LIN {X 0,Y 301.762,Z 448.822,A -85,B 0,C 180,E1 -16309.029,E2 -16309.029} C_VEL
LIN {X 0,Y 304.037,Z 439.587,A -85,B 0,C 180,E1 -16311.349,E2 -16311.349} C_VEL
LIN {X 0,Y 306.34,Z 429.711,A -85,B 0,C 180,E1 -16313.412,E2 -16313.412} C_VEL
LIN {X 0,Y 308.97,Z 418.014,A -85,B 0,C 180,E1 -16315.425,E2 -16315.425} C_VEL
LIN {X 0,Y 311.633,Z 405.588,A -85,B 0,C 180,E1 -16317.172,E2 -16317.172} C_VEL
LIN {X 0,Y 314.203,Z 392.482,A -85,B 0,C 180,E1 -16318.669,E2 -16318.669} C_VEL
LIN {X 0,Y 315.459,Z 385.45,A -85,B 0,C 180,E1 -16319.348,E2 -16319.348} C_VEL
LIN {X 0,Y 313.739,Z 373.355,A -85,B 0,C 180,E1 -16320.726,E2 -16320.726} C_VEL
LIN {X 0,Y 310.787,Z 359.836,A -85,B 0,C 180,E1 -16322.156,E2 -16322.156} C_VEL
LIN {X 0,Y 307.358,Z 347.749,A -85,B 0,C 180,E1 -16323.35,E2 -16323.35} C_VEL
LIN {X 0,Y 301.887,Z 332.55,A -85,B 0,C 180,E1 -16324.764,E2 -16324.764} C_VEL
LIN {X 0,Y 298.924,Z 325.57,A -85,B 0,C 180,E1 -16325.394,E2 -16325.394} C_VEL
LIN {X 0,Y 298.745,Z 324.598,A -85,B 0,C 180,E1 -16325.469,E2 -16325.469} C_VEL
LIN {X 0,Y 299.347,Z 320.548,A -85,B 0,C 180,E1 -16329.337,E2 -16329.337} C_VEL
LIN {X 0,Y 299.608,Z 317.074,A -85,B 0,C 180,E1 -16332.863,E2 -16332.863} C_VEL
LIN {X 0,Y 299.433,Z 314.897,A -85,B 0,C 180,E1 -16335.241,E2 -16335.241} C_VEL
LIN {X 0,Y 298.979,Z 311.805,A -85,B 0,C 180,E1 -16338.838,E2 -16338.838} C_VEL
LIN {X 0,Y 298.58,Z 309.054,A -85,B 0,C 180,E1 -16342.267,E2 -16342.267} C_VEL
LIN {X 0,Y 298.413,Z 307.944,A -85,B 0,C 180,E1 -16343.93,E2 -16343.93} C_VEL
LIN {X 0,Y 298.387,Z 307.95,A -85,B 0,C 180,E1 -16347.983,E2 -16347.983} C_VEL
LIN {X 0,Y 298.452,Z 307.939,A -85,B 0,C 180,E1 -16351.903,E2 -16351.903} C_VEL
LIN {X 0,Y 298.479,Z 307.931,A -85,B 0,C 180,E1 -16354.924,E2 -16354.924} C_VEL
LIN {X 0,Y 298.444,Z 307.935,A -85,B 0,C 180,E1 -16359.315,E2 -16359.315} C_VEL
LIN {X 0,Y 298.531,Z 307.922,A -85,B 0,C 180,E1 -16362.179,E2 -16362.179} C_VEL
LIN {X 0,Y 298.586,Z 307.914,A -85,B 0,C 180,E1 -16364.995,E2 -16364.995} C_VEL
LIN {X 0,Y 298.576,Z 307.918,A -85,B 0,C 180,E1 -16369.146,E2 -16369.146} C_VEL
LIN {X 0,Y 298.69,Z 307.902,A -85,B 0,C 180,E1 -16371.884,E2 -16371.884} C_VEL
LIN {X 0,Y 298.634,Z 307.907,A -85,B 0,C 180,E1 -16374.599,E2 -16374.599} C_VEL
LIN {X 0,Y 298.913,Z 307.875,A -85,B 0,C 180,E1 -16378.653,E2 -16378.653} C_VEL
LIN {X 0,Y 298.913,Z 307.878,A -85,B 0,C 180,E1 -16381.347,E2 -16381.347} C_VEL
LIN {X 0,Y 298.635,Z 307.911,A -85,B 0,C 180,E1 -16385.402,E2 -16385.402} C_VEL
LIN {X 0,Y 298.701,Z 307.898,A -85,B 0,C 180,E1 -16388.82,E2 -16388.82} C_VEL
LIN {X 0,Y 298.545,Z 307.924,A -85,B 0,C 180,E1 -16393.616,E2 -16393.616} C_VEL
LIN {X 0,Y 298.542,Z 307.923,A -85,B 0,C 180,E1 -16396.409,E2 -16396.409} C_VEL
LIN {X 0,Y 298.506,Z 307.928,A -85,B 0,C 180,E1 -16399.655,E2 -16399.655} C_VEL
LIN {X 0,Y 298.452,Z 307.934,A -85,B 0,C 180,E1 -16403.598,E2 -16403.598} C_VEL
LIN {X 0,Y 298.481,Z 307.928,A -85,B 0,C 180,E1 -16406.575,E2 -16406.575} C_VEL
LIN {X 0,Y 298.411,Z 307.935,A -85,B 0,C 180,E1 -16409.642,E2 -16409.642} C_VEL
LIN {X 0,Y 298.39,Z 307.937,A -85,B 0,C 180,E1 -16412.801,E2 -16412.801} C_VEL
LIN {X 0,Y 298.442,Z 307.934,A -85,B 0,C 180,E1 -16416.808,E2 -16416.808} C_VEL
LIN {X 0,Y 298.4,Z 307.942,A -85,B 0,C 180,E1 -16419.488,E2 -16419.488} C_VEL
LIN {X 0,Y 298.762,Z 310.457,A -85,B 0,C 180,E1 -16423.179,E2 -16423.179} C_VEL
LIN {X 0,Y 298.971,Z 311.975,A -85,B 0,C 180,E1 -16425.154,E2 -16425.154} C_VEL
LIN {X 0,Y 299.091,Z 315.034,A -85,B 0,C 180,E1 -16428.859,E2 -16428.859} C_VEL
LIN {X 0,Y 298.739,Z 318.083,A -85,B 0,C 180,E1 -16432.291,E2 -16432.291} C_VEL
LIN {X 0,Y 298.531,Z 320.183,A -85,B 0,C 180,E1 -16434.571,E2 -16434.571} C_VEL
LIN {X 0,Y 299.493,Z 323.226,A -85,B 0,C 180,E1 -16434.808,E2 -16434.808} C_VEL
LIN {X 0,Y 304.021,Z 333.557,A -85,B 0,C 180,E1 -16435.807,E2 -16435.807} C_VEL
LIN {X 0,Y 309.067,Z 347.625,A -85,B 0,C 180,E1 -16437.201,E2 -16437.201} C_VEL
LIN {X 0,Y 312.811,Z 361.239,A -85,B 0,C 180,E1 -16438.623,E2 -16438.623} C_VEL
LIN {X 0,Y 315.268,Z 373.146,A -85,B 0,C 180,E1 -16439.956,E2 -16439.956} C_VEL
LIN {X 0,Y 316.015,Z 378.195,A -85,B 0,C 180,E1 -16440.556,E2 -16440.556} C_VEL
LIN {X 0,Y 313.903,Z 390.512,A -85,B 0,C 180,E1 -16441.776,E2 -16441.776} C_VEL
LIN {X 0,Y 311.326,Z 403.463,A -85,B 0,C 180,E1 -16443.343,E2 -16443.343} C_VEL
LIN {X 0,Y 308.75,Z 415.307,A -85,B 0,C 180,E1 -16445.096,E2 -16445.096} C_VEL
LIN {X 0,Y 306.343,Z 426.145,A -85,B 0,C 180,E1 -16447.046,E2 -16447.046} C_VEL
LIN {X 0,Y 303.758,Z 436.69,A -85,B 0,C 180,E1 -16449.34,E2 -16449.34} C_VEL
LIN {X 0,Y 301.665,Z 445.456,A -85,B 0,C 180,E1 -16451.669,E2 -16451.669} C_VEL
LIN {X 0,Y 299.955,Z 452.887,A -85,B 0,C 180,E1 -16454.069,E2 -16454.069} C_VEL
LIN {X 0,Y 298.725,Z 458.754,A -85,B 0,C 180,E1 -16456.393,E2 -16456.393} C_VEL
LIN {X 0,Y 297.61,Z 464.23,A -85,B 0,C 180,E1 -16459.111,E2 -16459.111} C_VEL
LIN {X 0,Y 296.951,Z 468.363,A -85,B 0,C 180,E1 -16461.837,E2 -16461.837} C_VEL
LIN {X 0,Y 296.62,Z 471.267,A -85,B 0,C 180,E1 -16464.562,E2 -16464.562} C_VEL
LIN {X 0,Y 296.531,Z 473.012,A -85,B 0,C 180,E1 -16467.284,E2 -16467.284} C_VEL
LIN {X 0,Y 296.452,Z 473.621,A -85,B 0,C 180,E1 -16470.001,E2 -16470.001} C_VEL
LIN {X 0,Y 296.531,Z 473.052,A -85,B 0,C 180,E1 -16472.717,E2 -16472.717} C_VEL
LIN {X 0,Y 296.667,Z 471.11,A -85,B 0,C 180,E1 -16475.744,E2 -16475.744} C_VEL
LIN {X 0,Y 296.948,Z 468.508,A -85,B 0,C 180,E1 -16478.164,E2 -16478.164} C_VEL
LIN {X 0,Y 297.589,Z 464.424,A -85,B 0,C 180,E1 -16480.891,E2 -16480.891} C_VEL
LIN {X 0,Y 298.694,Z 459.01,A -85,B 0,C 180,E1 -16483.609,E2 -16483.609} C_VEL
LIN {X 0,Y 300.118,Z 452.113,A -85,B 0,C 180,E1 -16486.321,E2 -16486.321} C_VEL
LIN {X 0,Y 302.151,Z 443.505,A -85,B 0,C 180,E1 -16489.004,E2 -16489.004} C_VEL
LIN {X 0,Y 304.328,Z 434.355,A -85,B 0,C 180,E1 -16491.329,E2 -16491.329} C_VEL
LIN {X 0,Y 306.813,Z 424.173,A -85,B 0,C 180,E1 -16493.456,E2 -16493.456} C_VEL
LIN {X 0,Y 309.545,Z 411.912,A -85,B 0,C 180,E1 -16495.555,E2 -16495.555} C_VEL
LIN {X 0,Y 312.17,Z 399.379,A -85,B 0,C 180,E1 -16497.304,E2 -16497.304} C_VEL
LIN {X 0,Y 314.664,Z 387.068,A -85,B 0,C 180,E1 -16498.699,E2 -16498.699} C_VEL
LIN {X 0,Y 316.044,Z 379.083,A -85,B 0,C 180,E1 -16499.464,E2 -16499.464} C_VEL
LIN {X 0,Y 314.514,Z 368.782,A -85,B 0,C 180,E1 -16500.65,E2 -16500.65} C_VEL
LIN {X 0,Y 311.352,Z 355.334,A -85,B 0,C 180,E1 -16502.117,E2 -16502.117} C_VEL
LIN {X 0,Y 307,Z 341.307,A -85,B 0,C 180,E1 -16503.546,E2 -16503.546} C_VEL
LIN {X 0,Y 301.359,Z 327.255,A -85,B 0,C 180,E1 -16504.927,E2 -16504.927} C_VEL
LIN {X 0,Y 298.705,Z 321.182,A -85,B 0,C 180,E1 -16505.492,E2 -16505.492} C_VEL
LIN {X 0,Y 298.545,Z 320.158,A -85,B 0,C 180,E1 -16505.58,E2 -16505.58} C_VEL
LIN {X 0,Y 298.94,Z 316.682,A -85,B 0,C 180,E1 -16509.402,E2 -16509.402} C_VEL
LIN {X 0,Y 299.095,Z 315.081,A -85,B 0,C 180,E1 -16511.243,E2 -16511.243} C_VEL
LIN {X 0,Y 298.986,Z 312.099,A -85,B 0,C 180,E1 -16514.844,E2 -16514.844} C_VEL
LIN {X 0,Y 298.56,Z 309.055,A -85,B 0,C 180,E1 -16518.874,E2 -16518.874} C_VEL
LIN {X 0,Y 298.398,Z 307.943,A -85,B 0,C 180,E1 -16520.512,E2 -16520.512} C_VEL
LIN {X 0,Y 298.418,Z 307.942,A -85,B 0,C 180,E1 -16523.93,E2 -16523.93} C_VEL
LIN {X 0,Y 298.387,Z 307.944,A -85,B 0,C 180,E1 -16527.985,E2 -16527.985} C_VEL
LIN {X 0,Y 298.413,Z 307.939,A -85,B 0,C 180,E1 -16531.899,E2 -16531.899} C_VEL
LIN {X 0,Y 298.439,Z 307.935,A -85,B 0,C 180,E1 -16534.92,E2 -16534.92} C_VEL
LIN {X 0,Y 298.439,Z 307.936,A -85,B 0,C 180,E1 -16539.314,E2 -16539.314} C_VEL
LIN {X 0,Y 298.536,Z 307.924,A -85,B 0,C 180,E1 -16542.179,E2 -16542.179} C_VEL
LIN {X 0,Y 298.547,Z 307.918,A -85,B 0,C 180,E1 -16543.586,E2 -16543.586} C_VEL
LIN {X 0,Y 297.935,Z 307.998,A -85,B 0,C 180,E1 -16544.713,E2 -16544.713} C_VEL
LIN {X 0,Y 295.079,Z 308.355,A -85,B 0,C 180,E1 -16546.547,E2 -16546.547} C_VEL
LIN {X 0,Y 292.632,Z 308.658,A -85,B 0,C 180,E1 -16548.036,E2 -16548.036} C_VEL
LIN {X 0,Y 291.598,Z 308.789,A -85,B 0,C 180,E1 -16549.19,E2 -16549.19} C_VEL
LIN {X 0,Y 291.525,Z 308.794,A -85,B 0,C 180,E1 -16549.581,E2 -16549.581} C_VEL
LIN {X 0,Y 291.65,Z 308.78,A -85,B 0,C 180,E1 -16551.687,E2 -16551.687} C_VEL
LIN {X 0,Y 291.607,Z 308.787,A -85,B 0,C 180,E1 -16554.468,E2 -16554.468} C_VEL
LIN {X 0,Y 291.885,Z 308.753,A -85,B 0,C 180,E1 -16558.62,E2 -16558.62} C_VEL
LIN {X 0,Y 291.884,Z 308.752,A -85,B 0,C 180,E1 -16561.38,E2 -16561.38} C_VEL
LIN {X 0,Y 291.607,Z 308.786,A -85,B 0,C 180,E1 -16565.532,E2 -16565.532} C_VEL
LIN {X 0,Y 291.665,Z 308.779,A -85,B 0,C 180,E1 -16568.91,E2 -16568.91} C_VEL
LIN {X 0,Y 291.516,Z 308.799,A -85,B 0,C 180,E1 -16572.531,E2 -16572.531} C_VEL
LIN {X 0,Y 291.554,Z 308.795,A -85,B 0,C 180,E1 -16575.376,E2 -16575.376} C_VEL
LIN {X 0,Y 291.45,Z 308.808,A -85,B 0,C 180,E1 -16579.875,E2 -16579.875} C_VEL
LIN {X 0,Y 291.381,Z 308.815,A -85,B 0,C 180,E1 -16584.207,E2 -16584.207} C_VEL
LIN {X 0,Y 291.418,Z 308.813,A -85,B 0,C 180,E1 -16587.272,E2 -16587.272} C_VEL
LIN {X 0,Y 291.333,Z 308.827,A -85,B 0,C 180,E1 -16590.437,E2 -16590.437} C_VEL
LIN {X 0,Y 291.343,Z 308.829,A -85,B 0,C 180,E1 -16593.698,E2 -16593.698} C_VEL
LIN {X 0,Y 291.36,Z 308.828,A -85,B 0,C 180,E1 -16595.374,E2 -16595.374} C_VEL
LIN {X 0,Y 291.722,Z 311.173,A -85,B 0,C 180,E1 -16598.783,E2 -16598.783} C_VEL
LIN {X 0,Y 292.146,Z 314.013,A -85,B 0,C 180,E1 -16602.344,E2 -16602.344} C_VEL
LIN {X 0,Y 292.518,Z 317.273,A -85,B 0,C 180,E1 -16606.118,E2 -16606.118} C_VEL
LIN {X 0,Y 292.391,Z 320.487,A -85,B 0,C 180,E1 -16609.535,E2 -16609.535} C_VEL
LIN {X 0,Y 291.975,Z 323.962,A -85,B 0,C 180,E1 -16613.004,E2 -16613.004} C_VEL
LIN {X 0,Y 291.891,Z 324.512,A -85,B 0,C 180,E1 -16613.537,E2 -16613.537} C_VEL
LIN {X 0,Y 292.88,Z 327.696,A -85,B 0,C 180,E1 -16613.802,E2 -16613.802} C_VEL
LIN {X 0,Y 298.34,Z 340.78,A -85,B 0,C 180,E1 -16615.093,E2 -16615.093} C_VEL
LIN {X 0,Y 302.962,Z 355.274,A -85,B 0,C 180,E1 -16616.553,E2 -16616.553} C_VEL
LIN {X 0,Y 306.134,Z 368.142,A -85,B 0,C 180,E1 -16617.937,E2 -16617.937} C_VEL
LIN {X 0,Y 308.432,Z 381.307,A -85,B 0,C 180,E1 -16619.454,E2 -16619.454} C_VEL
LIN {X 0,Y 309.086,Z 386.746,A -85,B 0,C 180,E1 -16620.115,E2 -16620.115} C_VEL
LIN {X 0,Y 306.669,Z 399.186,A -85,B 0,C 180,E1 -16621.419,E2 -16621.419} C_VEL
LIN {X 0,Y 303.725,Z 412.723,A -85,B 0,C 180,E1 -16623.178,E2 -16623.178} C_VEL
LIN {X 0,Y 300.907,Z 424.901,A -85,B 0,C 180,E1 -16625.139,E2 -16625.139} C_VEL
LIN {X 0,Y 298.453,Z 435.156,A -85,B 0,C 180,E1 -16627.143,E2 -16627.143} C_VEL
LIN {X 0,Y 295.925,Z 445.11,A -85,B 0,C 180,E1 -16629.494,E2 -16629.494} C_VEL
LIN {X 0,Y 293.899,Z 453.404,A -85,B 0,C 180,E1 -16631.888,E2 -16631.888} C_VEL
LIN {X 0,Y 292.116,Z 461.195,A -85,B 0,C 180,E1 -16634.654,E2 -16634.654} C_VEL
LIN {X 0,Y 290.835,Z 467.392,A -85,B 0,C 180,E1 -16637.438,E2 -16637.438} C_VEL
LIN {X 0,Y 290.016,Z 472.185,A -85,B 0,C 180,E1 -16640.233,E2 -16640.233} C_VEL
LIN {X 0,Y 289.567,Z 475.696,A -85,B 0,C 180,E1 -16643.029,E2 -16643.029} C_VEL
LIN {X 0,Y 289.374,Z 478.005,A -85,B 0,C 180,E1 -16645.821,E2 -16645.821} C_VEL
LIN {X 0,Y 289.368,Z 479.166,A -85,B 0,C 180,E1 -16648.608,E2 -16648.608} C_VEL
LIN {X 0,Y 289.368,Z 479.163,A -85,B 0,C 180,E1 -16651.391,E2 -16651.391} C_VEL
LIN {X 0,Y 289.376,Z 477.989,A -85,B 0,C 180,E1 -16654.178,E2 -16654.178} C_VEL
LIN {X 0,Y 289.566,Z 475.67,A -85,B 0,C 180,E1 -16656.97,E2 -16656.97} C_VEL
LIN {X 0,Y 290.015,Z 472.154,A -85,B 0,C 180,E1 -16659.766,E2 -16659.766} C_VEL
LIN {X 0,Y 290.833,Z 467.353,A -85,B 0,C 180,E1 -16662.561,E2 -16662.561} C_VEL
LIN {X 0,Y 292.124,Z 461.135,A -85,B 0,C 180,E1 -16665.345,E2 -16665.345} C_VEL
LIN {X 0,Y 293.895,Z 453.328,A -85,B 0,C 180,E1 -16668.111,E2 -16668.111} C_VEL
LIN {X 0,Y 295.913,Z 445.024,A -85,B 0,C 180,E1 -16670.506,E2 -16670.506} C_VEL
LIN {X 0,Y 298.5,Z 435.019,A -85,B 0,C 180,E1 -16672.859,E2 -16672.859} C_VEL
LIN {X 0,Y 300.901,Z 424.786,A -85,B 0,C 180,E1 -16674.86,E2 -16674.86} C_VEL
LIN {X 0,Y 303.701,Z 412.587,A -85,B 0,C 180,E1 -16676.823,E2 -16676.823} C_VEL
LIN {X 0,Y 306.657,Z 399.002,A -85,B 0,C 180,E1 -16678.581,E2 -16678.581} C_VEL
LIN {X 0,Y 309.046,Z 386.658,A -85,B 0,C 180,E1 -16679.873,E2 -16679.873} C_VEL
LIN {X 0,Y 307.37,Z 374.793,A -85,B 0,C 180,E1 -16681.289,E2 -16681.289} C_VEL
LIN {X 0,Y 304.337,Z 360.53,A -85,B 0,C 180,E1 -16682.864,E2 -16682.864} C_VEL
LIN {X 0,Y 300.046,Z 345.896,A -85,B 0,C 180,E1 -16684.371,E2 -16684.371} C_VEL
LIN {X 0,Y 295.025,Z 332.512,A -85,B 0,C 180,E1 -16685.692,E2 -16685.692} C_VEL
LIN {X 0,Y 292.068,Z 325.637,A -85,B 0,C 180,E1 -16686.35,E2 -16686.35} C_VEL
LIN {X 0,Y 291.867,Z 324.527,A -85,B 0,C 180,E1 -16686.427,E2 -16686.427} C_VEL
LIN {X 0,Y 292.326,Z 321.204,A -85,B 0,C 180,E1 -16689.706,E2 -16689.706} C_VEL
LIN {X 0,Y 292.53,Z 318.735,A -85,B 0,C 180,E1 -16692.274,E2 -16692.274} C_VEL
LIN {X 0,Y 292.362,Z 315.557,A -85,B 0,C 180,E1 -16695.804,E2 -16695.804} C_VEL
LIN {X 0,Y 291.889,Z 312.541,A -85,B 0,C 180,E1 -16699.451,E2 -16699.451} C_VEL
LIN {X 0,Y 291.521,Z 309.849,A -85,B 0,C 180,E1 -16702.937,E2 -16702.937} C_VEL
LIN {X 0,Y 291.356,Z 308.824,A -85,B 0,C 180,E1 -16704.625,E2 -16704.625} C_VEL
LIN {X 0,Y 291.364,Z 308.825,A -85,B 0,C 180,E1 -16707.95,E2 -16707.95} C_VEL
LIN {X 0,Y 291.371,Z 308.82,A -85,B 0,C 180,E1 -16711.157,E2 -16711.157} C_VEL
LIN {X 0,Y 291.41,Z 308.812,A -85,B 0,C 180,E1 -16714.271,E2 -16714.271} C_VEL
LIN {X 0,Y 291.375,Z 308.817,A -85,B 0,C 180,E1 -16717.299,E2 -16717.299} C_VEL
LIN {X 0,Y 291.452,Z 308.804,A -85,B 0,C 180,E1 -16720.27,E2 -16720.27} C_VEL
LIN {X 0,Y 291.534,Z 308.794,A -85,B 0,C 180,E1 -16724.634,E2 -16724.634} C_VEL
LIN {X 0,Y 291.522,Z 308.796,A -85,B 0,C 180,E1 -16728.88,E2 -16728.88} C_VEL
LIN {X 0,Y 291.644,Z 308.78,A -85,B 0,C 180,E1 -16731.687,E2 -16731.687} C_VEL
LIN {X 0,Y 291.602,Z 308.783,A -85,B 0,C 180,E1 -16734.468,E2 -16734.468} C_VEL
LIN {X 0,Y 291.88,Z 308.751,A -85,B 0,C 180,E1 -16738.62,E2 -16738.62} C_VEL
LIN {X 0,Y 291.88,Z 308.754,A -85,B 0,C 180,E1 -16741.38,E2 -16741.38} C_VEL
LIN {X 0,Y 291.642,Z 308.78,A -85,B 0,C 180,E1 -16746.533,E2 -16746.533} C_VEL
LIN {X 0,Y 291.561,Z 308.793,A -85,B 0,C 180,E1 -16749.714,E2 -16749.714} C_VEL
LIN {X 0,Y 291.515,Z 308.796,A -85,B 0,C 180,E1 -16753.951,E2 -16753.951} C_VEL
LIN {X 0,Y 291.481,Z 308.802,A -85,B 0,C 180,E1 -16756.818,E2 -16756.818} C_VEL
LIN {X 0,Y 291.445,Z 308.806,A -85,B 0,C 180,E1 -16759.875,E2 -16759.875} C_VEL
LIN {X 0,Y 291.395,Z 308.814,A -85,B 0,C 180,E1 -16764.206,E2 -16764.206} C_VEL
LIN {X 0,Y 291.414,Z 308.808,A -85,B 0,C 180,E1 -16767.273,E2 -16767.273} C_VEL
LIN {X 0,Y 291.329,Z 308.817,A -85,B 0,C 180,E1 -16770.438,E2 -16770.438} C_VEL
LIN {X 0,Y 291.339,Z 308.816,A -85,B 0,C 180,E1 -16773.699,E2 -16773.699} C_VEL
LIN {X 0,Y 291.371,Z 308.815,A -85,B 0,C 180,E1 -16777.255,E2 -16777.255} C_VEL
LIN {X 0,Y 291.398,Z 309.016,A -85,B 0,C 180,E1 -16779.488,E2 -16779.488} C_VEL
LIN {X 0,Y 291.808,Z 312.06,A -85,B 0,C 180,E1 -16783.738,E2 -16783.738} C_VEL
LIN {X 0,Y 292.004,Z 313.967,A -85,B 0,C 180,E1 -16786.224,E2 -16786.224} C_VEL
LIN {X 0,Y 292.003,Z 316.637,A -85,B 0,C 180,E1 -16789.472,E2 -16789.472} C_VEL
LIN {X 0,Y 291.615,Z 320.296,A -85,B 0,C 180,E1 -16793.606,E2 -16793.606} C_VEL
LIN {X 0,Y 292.49,Z 323.161,A -85,B 0,C 180,E1 -16793.829,E2 -16793.829} C_VEL
LIN {X 0,Y 293.765,Z 325.811,A -85,B 0,C 180,E1 -16794.104,E2 -16794.104} C_VEL
LIN {X 0,Y 299.181,Z 338.663,A -85,B 0,C 180,E1 -16795.426,E2 -16795.426} C_VEL
LIN {X 0,Y 303.595,Z 351.639,A -85,B 0,C 180,E1 -16796.792,E2 -16796.792} C_VEL
LIN {X 0,Y 307.308,Z 366.226,A -85,B 0,C 180,E1 -16798.417,E2 -16798.417} C_VEL
LIN {X 0,Y 309.462,Z 378.455,A -85,B 0,C 180,E1 -16799.888,E2 -16799.888} C_VEL
LIN {X 0,Y 309.443,Z 381.11,A -85,B 0,C 180,E1 -16800.175,E2 -16800.175} C_VEL
LIN {X 0,Y 306.792,Z 394.787,A -85,B 0,C 180,E1 -16801.62,E2 -16801.62} C_VEL
LIN {X 0,Y 304.255,Z 407.042,A -85,B 0,C 180,E1 -16803.23,E2 -16803.23} C_VEL
LIN {X 0,Y 301.43,Z 419.251,A -85,B 0,C 180,E1 -16805.187,E2 -16805.187} C_VEL
LIN {X 0,Y 298.988,Z 429.465,A -85,B 0,C 180,E1 -16807.18,E2 -16807.18} C_VEL
LIN {X 0,Y 296.42,Z 439.461,A -85,B 0,C 180,E1 -16809.531,E2 -16809.531} C_VEL
LIN {X 0,Y 294.303,Z 447.752,A -85,B 0,C 180,E1 -16811.915,E2 -16811.915} C_VEL
LIN {X 0,Y 292.733,Z 454.42,A -85,B 0,C 180,E1 -16814.245,E2 -16814.245} C_VEL
LIN {X 0,Y 291.435,Z 460.32,A -85,B 0,C 180,E1 -16816.757,E2 -16816.757} C_VEL
LIN {X 0,Y 290.398,Z 465.467,A -85,B 0,C 180,E1 -16819.543,E2 -16819.543} C_VEL
LIN {X 0,Y 289.895,Z 468.433,A -85,B 0,C 180,E1 -16821.637,E2 -16821.637} C_VEL
LIN {X 0,Y 289.556,Z 471.336,A -85,B 0,C 180,E1 -16824.429,E2 -16824.429} C_VEL
LIN {X 0,Y 289.437,Z 473.081,A -85,B 0,C 180,E1 -16827.217,E2 -16827.217} C_VEL
LIN {X 0,Y 289.372,Z 473.69,A -85,B 0,C 180,E1 -16830.001,E2 -16830.001} C_VEL
LIN {X 0,Y 289.437,Z 473.121,A -85,B 0,C 180,E1 -16832.784,E2 -16832.784} C_VEL
LIN {X 0,Y 289.587,Z 471.317,A -85,B 0,C 180,E1 -16835.713,E2 -16835.713} C_VEL
LIN {X 0,Y 289.892,Z 468.577,A -85,B 0,C 180,E1 -16838.364,E2 -16838.364} C_VEL
LIN {X 0,Y 290.571,Z 464.492,A -85,B 0,C 180,E1 -16841.157,E2 -16841.157} C_VEL
LIN {X 0,Y 291.752,Z 459.078,A -85,B 0,C 180,E1 -16843.939,E2 -16843.939} C_VEL
LIN {X 0,Y 293.25,Z 452.181,A -85,B 0,C 180,E1 -16846.714,E2 -16846.714} C_VEL
LIN {X 0,Y 295.385,Z 443.573,A -85,B 0,C 180,E1 -16849.457,E2 -16849.457} C_VEL
LIN {X 0,Y 297.701,Z 434.422,A -85,B 0,C 180,E1 -16851.828,E2 -16851.828} C_VEL
LIN {X 0,Y 300.112,Z 424.883,A -85,B 0,C 180,E1 -16853.875,E2 -16853.875} C_VEL
LIN {X 0,Y 302.884,Z 413.041,A -85,B 0,C 180,E1 -16855.974,E2 -16855.974} C_VEL
LIN {X 0,Y 305.616,Z 400.724,A -85,B 0,C 180,E1 -16857.754,E2 -16857.754} C_VEL
LIN {X 0,Y 308.372,Z 387.5,A -85,B 0,C 180,E1 -16859.296,E2 -16859.296} C_VEL
LIN {X 0,Y 309.582,Z 380.809,A -85,B 0,C 180,E1 -16859.963,E2 -16859.963} C_VEL
LIN {X 0,Y 309.141,Z 376.231,A -85,B 0,C 180,E1 -16860.503,E2 -16860.503} C_VEL
LIN {X 0,Y 306.677,Z 363.447,A -85,B 0,C 180,E1 -16862.014,E2 -16862.014} C_VEL
LIN {X 0,Y 303.174,Z 350.218,A -85,B 0,C 180,E1 -16863.474,E2 -16863.474} C_VEL
LIN {X 0,Y 298.502,Z 336.794,A -85,B 0,C 180,E1 -16864.892,E2 -16864.892} C_VEL
LIN {X 0,Y 292.91,Z 323.875,A -85,B 0,C 180,E1 -16866.212,E2 -16866.212} C_VEL
LIN {X 0,Y 291.78,Z 321.283,A -85,B 0,C 180,E1 -16866.466,E2 -16866.466} C_VEL
LIN {X 0,Y 291.587,Z 320.238,A -85,B 0,C 180,E1 -16866.567,E2 -16866.567} C_VEL
LIN {X 0,Y 292.007,Z 316.769,A -85,B 0,C 180,E1 -16870.529,E2 -16870.529} C_VEL
LIN {X 0,Y 292.011,Z 313.698,A -85,B 0,C 180,E1 -16874.263,E2 -16874.263} C_VEL
LIN {X 0,Y 291.684,Z 311.211,A -85,B 0,C 180,E1 -16877.573,E2 -16877.573} C_VEL
LIN {X 0,Y 291.351,Z 308.821,A -85,B 0,C 180,E1 -16881.158,E2 -16881.158} C_VEL
LIN {X 0,Y 291.361,Z 308.82,A -85,B 0,C 180,E1 -16884.626,E2 -16884.626} C_VEL
LIN {X 0,Y 291.365,Z 308.818,A -85,B 0,C 180,E1 -16887.95,E2 -16887.95} C_VEL
LIN {X 0,Y 291.343,Z 308.819,A -85,B 0,C 180,E1 -16891.154,E2 -16891.154} C_VEL
LIN {X 0,Y 291.359,Z 308.819,A -85,B 0,C 180,E1 -16894.266,E2 -16894.266} C_VEL
LIN {X 0,Y 291.371,Z 308.814,A -85,B 0,C 180,E1 -16897.298,E2 -16897.298} C_VEL
LIN {X 0,Y 291.457,Z 308.802,A -85,B 0,C 180,E1 -16900.27,E2 -16900.27} C_VEL
LIN {X 0,Y 291.555,Z 308.791,A -85,B 0,C 180,E1 -16904.624,E2 -16904.624} C_VEL
LIN {X 0,Y 291.527,Z 308.797,A -85,B 0,C 180,E1 -16908.88,E2 -16908.88} C_VEL
LIN {X 0,Y 291.525,Z 308.794,A -85,B 0,C 180,E1 -16909.581,E2 -16909.581} C_VEL
LIN {X 0,Y 290.885,Z 308.878,A -85,B 0,C 180,E1 -16910.735,E2 -16910.735} C_VEL
LIN {X 0,Y 288.039,Z 309.232,A -85,B 0,C 180,E1 -16912.615,E2 -16912.615} C_VEL
LIN {X 0,Y 285.613,Z 309.535,A -85,B 0,C 180,E1 -16914.141,E2 -16914.141} C_VEL
LIN {X 0,Y 284.579,Z 309.662,A -85,B 0,C 180,E1 -16915.323,E2 -16915.323} C_VEL
LIN {X 0,Y 284.499,Z 309.672,A -85,B 0,C 180,E1 -16915.724,E2 -16915.724} C_VEL
LIN {X 0,Y 284.852,Z 309.629,A -85,B 0,C 180,E1 -16918.586,E2 -16918.586} C_VEL
LIN {X 0,Y 284.851,Z 309.628,A -85,B 0,C 180,E1 -16921.414,E2 -16921.414} C_VEL
LIN {X 0,Y 284.575,Z 309.662,A -85,B 0,C 180,E1 -16925.669,E2 -16925.669} C_VEL
LIN {X 0,Y 284.606,Z 309.659,A -85,B 0,C 180,E1 -16928.98,E2 -16928.98} C_VEL
LIN {X 0,Y 284.473,Z 309.676,A -85,B 0,C 180,E1 -16932.847,E2 -16932.847} C_VEL
LIN {X 0,Y 284.486,Z 309.674,A -85,B 0,C 180,E1 -16935.768,E2 -16935.768} C_VEL
LIN {X 0,Y 284.376,Z 309.688,A -85,B 0,C 180,E1 -16940.242,E2 -16940.242} C_VEL
LIN {X 0,Y 284.336,Z 309.692,A -85,B 0,C 180,E1 -16944.847,E2 -16944.847} C_VEL
LIN {X 0,Y 284.327,Z 309.696,A -85,B 0,C 180,E1 -16948.011,E2 -16948.011} C_VEL
LIN {X 0,Y 284.292,Z 309.705,A -85,B 0,C 180,E1 -16951.275,E2 -16951.275} C_VEL
LIN {X 0,Y 284.308,Z 309.706,A -85,B 0,C 180,E1 -16954.649,E2 -16954.649} C_VEL
LIN {X 0,Y 284.66,Z 311.954,A -85,B 0,C 180,E1 -16958.114,E2 -16958.114} C_VEL
LIN {X 0,Y 285.148,Z 315.206,A -85,B 0,C 180,E1 -16962.32,E2 -16962.32} C_VEL
LIN {X 0,Y 285.476,Z 317.895,A -85,B 0,C 180,E1 -16965.556,E2 -16965.556} C_VEL
LIN {X 0,Y 285.461,Z 320.418,A -85,B 0,C 180,E1 -16968.338,E2 -16968.338} C_VEL
LIN {X 0,Y 285.079,Z 324.014,A -85,B 0,C 180,E1 -16972.082,E2 -16972.082} C_VEL
LIN {X 0,Y 285.04,Z 324.631,A -85,B 0,C 180,E1 -16972.536,E2 -16972.536} C_VEL
LIN {X 0,Y 286.07,Z 327.739,A -85,B 0,C 180,E1 -16972.801,E2 -16972.801} C_VEL
LIN {X 0,Y 287.425,Z 330.751,A -85,B 0,C 180,E1 -16973.115,E2 -16973.115} C_VEL
LIN {X 0,Y 293.007,Z 344.703,A -85,B 0,C 180,E1 -16974.586,E2 -16974.586} C_VEL
LIN {X 0,Y 297.212,Z 358.54,A -85,B 0,C 180,E1 -16976.064,E2 -16976.064} C_VEL
LIN {X 0,Y 300.11,Z 370.919,A -85,B 0,C 180,E1 -16977.463,E2 -16977.463} C_VEL
LIN {X 0,Y 302.178,Z 383.779,A -85,B 0,C 180,E1 -16979.031,E2 -16979.031} C_VEL
LIN {X 0,Y 302.642,Z 387.691,A -85,B 0,C 180,E1 -16979.534,E2 -16979.534} C_VEL
LIN {X 0,Y 300.137,Z 400.444,A -85,B 0,C 180,E1 -16980.93,E2 -16980.93} C_VEL
LIN {X 0,Y 297.397,Z 412.657,A -85,B 0,C 180,E1 -16982.56,E2 -16982.56} C_VEL
LIN {X 0,Y 294.428,Z 424.834,A -85,B 0,C 180,E1 -16984.554,E2 -16984.554} C_VEL
LIN {X 0,Y 291.787,Z 435.391,A -85,B 0,C 180,E1 -16986.663,E2 -16986.663} C_VEL
LIN {X 0,Y 289.205,Z 445.042,A -85,B 0,C 180,E1 -16988.995,E2 -16988.995} C_VEL
LIN {X 0,Y 287.112,Z 453.336,A -85,B 0,C 180,E1 -16991.445,E2 -16991.445} C_VEL
LIN {X 0,Y 285.19,Z 461.126,A -85,B 0,C 180,E1 -16994.271,E2 -16994.271} C_VEL
LIN {X 0,Y 283.874,Z 467.324,A -85,B 0,C 180,E1 -16997.125,E2 -16997.125} C_VEL
LIN {X 0,Y 282.971,Z 472.116,A -85,B 0,C 180,E1 -16999.988,E2 -16999.988} C_VEL
LIN {X 0,Y 282.487,Z 475.627,A -85,B 0,C 180,E1 -17002.854,E2 -17002.854} C_VEL
LIN {X 0,Y 282.284,Z 477.936,A -85,B 0,C 180,E1 -17005.716,E2 -17005.716} C_VEL
LIN {X 0,Y 282.293,Z 479.097,A -85,B 0,C 180,E1 -17008.573,E2 -17008.573} C_VEL
LIN {X 0,Y 282.293,Z 479.094,A -85,B 0,C 180,E1 -17011.426,E2 -17011.426} C_VEL
LIN {X 0,Y 282.286,Z 477.92,A -85,B 0,C 180,E1 -17014.283,E2 -17014.283} C_VEL
LIN {X 0,Y 282.487,Z 475.6,A -85,B 0,C 180,E1 -17017.145,E2 -17017.145} C_VEL
LIN {X 0,Y 282.97,Z 472.084,A -85,B 0,C 180,E1 -17020.011,E2 -17020.011} C_VEL
LIN {X 0,Y 283.872,Z 467.282,A -85,B 0,C 180,E1 -17022.874,E2 -17022.874} C_VEL
LIN {X 0,Y 285.197,Z 461.064,A -85,B 0,C 180,E1 -17025.727,E2 -17025.727} C_VEL
LIN {X 0,Y 287.106,Z 453.256,A -85,B 0,C 180,E1 -17028.555,E2 -17028.555} C_VEL
LIN {X 0,Y 289.198,Z 444.952,A -85,B 0,C 180,E1 -17031.004,E2 -17031.004} C_VEL
LIN {X 0,Y 291.866,Z 435.101,A -85,B 0,C 180,E1 -17033.373,E2 -17033.373} C_VEL
LIN {X 0,Y 294.419,Z 424.714,A -85,B 0,C 180,E1 -17035.446,E2 -17035.446} C_VEL
LIN {X 0,Y 297.357,Z 412.515,A -85,B 0,C 180,E1 -17037.443,E2 -17037.443} C_VEL
LIN {X 0,Y 300.423,Z 398.928,A -85,B 0,C 180,E1 -17039.231,E2 -17039.231} C_VEL
LIN {X 0,Y 302.571,Z 387.799,A -85,B 0,C 180,E1 -17040.431,E2 -17040.431} C_VEL
LIN {X 0,Y 300.818,Z 375.352,A -85,B 0,C 180,E1 -17041.987,E2 -17041.987} C_VEL
LIN {X 0,Y 298.205,Z 362.464,A -85,B 0,C 180,E1 -17043.472,E2 -17043.472} C_VEL
LIN {X 0,Y 294.034,Z 348.026,A -85,B 0,C 180,E1 -17045.05,E2 -17045.05} C_VEL
LIN {X 0,Y 289.483,Z 335.708,A -85,B 0,C 180,E1 -17046.339,E2 -17046.339} C_VEL
LIN {X 0,Y 285.967,Z 327.591,A -85,B 0,C 180,E1 -17047.181,E2 -17047.181} C_VEL
LIN {X 0,Y 284.978,Z 324.45,A -85,B 0,C 180,E1 -17047.452,E2 -17047.452} C_VEL
LIN {X 0,Y 285.341,Z 321.744,A -85,B 0,C 180,E1 -17050.223,E2 -17050.223} C_VEL
LIN {X 0,Y 285.486,Z 318.652,A -85,B 0,C 180,E1 -17053.573,E2 -17053.573} C_VEL
LIN {X 0,Y 285.296,Z 316.232,A -85,B 0,C 180,E1 -17056.39,E2 -17056.39} C_VEL
LIN {X 0,Y 284.825,Z 313.279,A -85,B 0,C 180,E1 -17060.093,E2 -17060.093} C_VEL
LIN {X 0,Y 284.433,Z 310.657,A -85,B 0,C 180,E1 -17063.629,E2 -17063.629} C_VEL
LIN {X 0,Y 284.303,Z 309.703,A -85,B 0,C 180,E1 -17065.35,E2 -17065.35} C_VEL
LIN {X 0,Y 284.288,Z 309.706,A -85,B 0,C 180,E1 -17068.725,E2 -17068.725} C_VEL
LIN {X 0,Y 284.39,Z 309.688,A -85,B 0,C 180,E1 -17072.826,E2 -17072.826} C_VEL
LIN {X 0,Y 284.36,Z 309.689,A -85,B 0,C 180,E1 -17076.707,E2 -17076.707} C_VEL
LIN {X 0,Y 284.397,Z 309.685,A -85,B 0,C 180,E1 -17081.261,E2 -17081.261} C_VEL
LIN {X 0,Y 284.472,Z 309.675,A -85,B 0,C 180,E1 -17084.469,E2 -17084.469} C_VEL
LIN {X 0,Y 284.476,Z 309.673,A -85,B 0,C 180,E1 -17088.601,E2 -17088.601} C_VEL
LIN {X 0,Y 284.601,Z 309.656,A -85,B 0,C 180,E1 -17091.48,E2 -17091.48} C_VEL
LIN {X 0,Y 284.571,Z 309.658,A -85,B 0,C 180,E1 -17094.331,E2 -17094.331} C_VEL
LIN {X 0,Y 284.846,Z 309.626,A -85,B 0,C 180,E1 -17098.586,E2 -17098.586} C_VEL
LIN {X 0,Y 284.846,Z 309.631,A -85,B 0,C 180,E1 -17101.414,E2 -17101.414} C_VEL
LIN {X 0,Y 284.591,Z 309.658,A -85,B 0,C 180,E1 -17106.55,E2 -17106.55} C_VEL
LIN {X 0,Y 284.507,Z 309.671,A -85,B 0,C 180,E1 -17109.958,E2 -17109.958} C_VEL
LIN {X 0,Y 284.472,Z 309.672,A -85,B 0,C 180,E1 -17114.303,E2 -17114.303} C_VEL
LIN {X 0,Y 284.419,Z 309.679,A -85,B 0,C 180,E1 -17117.249,E2 -17117.249} C_VEL
LIN {X 0,Y 284.373,Z 309.685,A -85,B 0,C 180,E1 -17120.243,E2 -17120.243} C_VEL
LIN {X 0,Y 284.364,Z 309.689,A -85,B 0,C 180,E1 -17123.876,E2 -17123.876} C_VEL
LIN {X 0,Y 284.39,Z 309.683,A -85,B 0,C 180,E1 -17127.173,E2 -17127.173} C_VEL
LIN {X 0,Y 284.288,Z 309.693,A -85,B 0,C 180,E1 -17131.275,E2 -17131.275} C_VEL
LIN {X 0,Y 284.336,Z 309.69,A -85,B 0,C 180,E1 -17135.349,E2 -17135.349} C_VEL
LIN {X 0,Y 284.308,Z 309.696,A -85,B 0,C 180,E1 -17138.17,E2 -17138.17} C_VEL
LIN {X 0,Y 284.462,Z 310.622,A -85,B 0,C 180,E1 -17140.015,E2 -17140.015} C_VEL
LIN {X 0,Y 284.892,Z 313.663,A -85,B 0,C 180,E1 -17144.326,E2 -17144.326} C_VEL
LIN {X 0,Y 285.029,Z 316.265,A -85,B 0,C 180,E1 -17147.707,E2 -17147.707} C_VEL
LIN {X 0,Y 284.909,Z 318.241,A -85,B 0,C 180,E1 -17150.109,E2 -17150.109} C_VEL
LIN {X 0,Y 284.673,Z 320.33,A -85,B 0,C 180,E1 -17152.544,E2 -17152.544} C_VEL
LIN {X 0,Y 285.746,Z 323.552,A -85,B 0,C 180,E1 -17152.844,E2 -17152.844} C_VEL
LIN {X 0,Y 286.889,Z 325.864,A -85,B 0,C 180,E1 -17153.102,E2 -17153.102} C_VEL
LIN {X 0,Y 292.238,Z 338.283,A -85,B 0,C 180,E1 -17154.454,E2 -17154.454} C_VEL
LIN {X 0,Y 296.909,Z 351.708,A -85,B 0,C 180,E1 -17155.942,E2 -17155.942} C_VEL
LIN {X 0,Y 300.268,Z 364.555,A -85,B 0,C 180,E1 -17157.431,E2 -17157.431} C_VEL
LIN {X 0,Y 302.439,Z 375.613,A -85,B 0,C 180,E1 -17158.79,E2 -17158.79} C_VEL
LIN {X 0,Y 303.238,Z 381.101,A -85,B 0,C 180,E1 -17159.491,E2 -17159.491} C_VEL
LIN {X 0,Y 300.553,Z 394.86,A -85,B 0,C 180,E1 -17160.975,E2 -17160.975} C_VEL
LIN {X 0,Y 297.913,Z 407.115,A -85,B 0,C 180,E1 -17162.613,E2 -17162.613} C_VEL
LIN {X 0,Y 294.957,Z 419.324,A -85,B 0,C 180,E1 -17164.604,E2 -17164.604} C_VEL
LIN {X 0,Y 292.412,Z 429.538,A -85,B 0,C 180,E1 -17166.637,E2 -17166.637} C_VEL
LIN {X 0,Y 289.741,Z 439.533,A -85,B 0,C 180,E1 -17169.037,E2 -17169.037} C_VEL
LIN {X 0,Y 287.513,Z 447.824,A -85,B 0,C 180,E1 -17171.473,E2 -17171.473} C_VEL
LIN {X 0,Y 285.58,Z 455.611,A -85,B 0,C 180,E1 -17174.295,E2 -17174.295} C_VEL
LIN {X 0,Y 284.111,Z 461.81,A -85,B 0,C 180,E1 -17177.137,E2 -17177.137} C_VEL
LIN {X 0,Y 283.187,Z 466.597,A -85,B 0,C 180,E1 -17179.996,E2 -17179.996} C_VEL
LIN {X 0,Y 282.599,Z 470.103,A -85,B 0,C 180,E1 -17182.858,E2 -17182.858} C_VEL
LIN {X 0,Y 282.359,Z 472.42,A -85,B 0,C 180,E1 -17185.718,E2 -17185.718} C_VEL
LIN {X 0,Y 282.307,Z 473.601,A -85,B 0,C 180,E1 -17188.574,E2 -17188.574} C_VEL
LIN {X 0,Y 282.307,Z 473.614,A -85,B 0,C 180,E1 -17191.427,E2 -17191.427} C_VEL
LIN {X 0,Y 282.359,Z 472.487,A -85,B 0,C 180,E1 -17194.283,E2 -17194.283} C_VEL
LIN {X 0,Y 282.599,Z 470.221,A -85,B 0,C 180,E1 -17197.143,E2 -17197.143} C_VEL
LIN {X 0,Y 283.171,Z 466.762,A -85,B 0,C 180,E1 -17200.005,E2 -17200.005} C_VEL
LIN {X 0,Y 284.091,Z 462.028,A -85,B 0,C 180,E1 -17202.865,E2 -17202.865} C_VEL
LIN {X 0,Y 285.521,Z 455.895,A -85,B 0,C 180,E1 -17205.71,E2 -17205.71} C_VEL
LIN {X 0,Y 287.461,Z 448.175,A -85,B 0,C 180,E1 -17208.532,E2 -17208.532} C_VEL
LIN {X 0,Y 289.65,Z 439.945,A -85,B 0,C 180,E1 -17210.971,E2 -17210.971} C_VEL
LIN {X 0,Y 292.34,Z 430.032,A -85,B 0,C 180,E1 -17213.37,E2 -17213.37} C_VEL
LIN {X 0,Y 294.856,Z 419.871,A -85,B 0,C 180,E1 -17215.407,E2 -17215.407} C_VEL
LIN {X 0,Y 297.54,Z 408.84,A -85,B 0,C 180,E1 -17217.235,E2 -17217.235} C_VEL
LIN {X 0,Y 300.134,Z 396.931,A -85,B 0,C 180,E1 -17218.879,E2 -17218.879} C_VEL
LIN {X 0,Y 302.839,Z 383.937,A -85,B 0,C 180,E1 -17220.327,E2 -17220.327} C_VEL
LIN {X 0,Y 303.21,Z 380.875,A -85,B 0,C 180,E1 -17220.659,E2 -17220.659} C_VEL
LIN {X 0,Y 301.13,Z 368.444,A -85,B 0,C 180,E1 -17222.219,E2 -17222.219} C_VEL
LIN {X 0,Y 297.905,Z 355.325,A -85,B 0,C 180,E1 -17223.767,E2 -17223.767} C_VEL
LIN {X 0,Y 293.737,Z 342.173,A -85,B 0,C 180,E1 -17225.236,E2 -17225.236} C_VEL
LIN {X 0,Y 288.061,Z 328.262,A -85,B 0,C 180,E1 -17226.763,E2 -17226.763} C_VEL
LIN {X 0,Y 285.756,Z 323.583,A -85,B 0,C 180,E1 -17227.282,E2 -17227.282} C_VEL
LIN {X 0,Y 284.665,Z 320.339,A -85,B 0,C 180,E1 -17227.587,E2 -17227.587} C_VEL
LIN {X 0,Y 284.945,Z 318.164,A -85,B 0,C 180,E1 -17230.129,E2 -17230.129} C_VEL
LIN {X 0,Y 285.042,Z 315.305,A -85,B 0,C 180,E1 -17233.659,E2 -17233.659} C_VEL
LIN {X 0,Y 284.82,Z 313.325,A -85,B 0,C 180,E1 -17236.298,E2 -17236.298} C_VEL
LIN {X 0,Y 284.45,Z 310.702,A -85,B 0,C 180,E1 -17240.03,E2 -17240.03} C_VEL
LIN {X 0,Y 284.322,Z 309.697,A -85,B 0,C 180,E1 -17242.278,E2 -17242.278} C_VEL
LIN {X 0,Y 284.308,Z 309.7,A -85,B 0,C 180,E1 -17245.351,E2 -17245.351} C_VEL
LIN {X 0,Y 284.284,Z 309.701,A -85,B 0,C 180,E1 -17248.724,E2 -17248.724} C_VEL
LIN {X 0,Y 284.283,Z 309.699,A -85,B 0,C 180,E1 -17251.984,E2 -17251.984} C_VEL
LIN {X 0,Y 284.32,Z 309.695,A -85,B 0,C 180,E1 -17256.146,E2 -17256.146} C_VEL
LIN {X 0,Y 284.387,Z 309.685,A -85,B 0,C 180,E1 -17259.898,E2 -17259.898} C_VEL
LIN {X 0,Y 284.491,Z 309.67,A -85,B 0,C 180,E1 -17264.459,E2 -17264.459} C_VEL
LIN {X 0,Y 284.481,Z 309.674,A -85,B 0,C 180,E1 -17268.601,E2 -17268.601} C_VEL
LIN {X 0,Y 284.607,Z 309.657,A -85,B 0,C 180,E1 -17271.479,E2 -17271.479} C_VEL
LIN {X 0,Y 284.575,Z 309.663,A -85,B 0,C 180,E1 -17274.331,E2 -17274.331} C_VEL
LIN {X 0,Y 284.499,Z 309.672,A -85,B 0,C 180,E1 -17275.724,E2 -17275.724} C_VEL
LIN {X 0,Y 283.889,Z 309.754,A -85,B 0,C 180,E1 -17276.908,E2 -17276.908} C_VEL
LIN {X 0,Y 281.215,Z 310.087,A -85,B 0,C 180,E1 -17278.844,E2 -17278.844} C_VEL
LIN {X 0,Y 278.102,Z 310.469,A -85,B 0,C 180,E1 -17281.219,E2 -17281.219} C_VEL
LIN {X 0,Y 277.746,Z 310.51,A -85,B 0,C 180,E1 -17282.038,E2 -17282.038} C_VEL
LIN {X 0,Y 277.6,Z 310.531,A -85,B 0,C 180,E1 -17287.272,E2 -17287.272} C_VEL
LIN {X 0,Y 277.456,Z 310.55,A -85,B 0,C 180,E1 -17290.213,E2 -17290.213} C_VEL
LIN {X 0,Y 277.433,Z 310.553,A -85,B 0,C 180,E1 -17294.674,E2 -17294.674} C_VEL
LIN {X 0,Y 277.341,Z 310.563,A -85,B 0,C 180,E1 -17299.234,E2 -17299.234} C_VEL
LIN {X 0,Y 277.291,Z 310.57,A -85,B 0,C 180,E1 -17304.157,E2 -17304.157} C_VEL
LIN {X 0,Y 277.322,Z 310.569,A -85,B 0,C 180,E1 -17307.504,E2 -17307.504} C_VEL
LIN {X 0,Y 277.271,Z 310.578,A -85,B 0,C 180,E1 -17310.481,E2 -17310.481} C_VEL
LIN {X 0,Y 277.246,Z 310.585,A -85,B 0,C 180,E1 -17313.896,E2 -17313.896} C_VEL
LIN {X 0,Y 277.587,Z 312.746,A -85,B 0,C 180,E1 -17317.419,E2 -17317.419} C_VEL
LIN {X 0,Y 277.986,Z 315.446,A -85,B 0,C 180,E1 -17321.096,E2 -17321.096} C_VEL
LIN {X 0,Y 278.419,Z 318.597,A -85,B 0,C 180,E1 -17325.026,E2 -17325.026} C_VEL
LIN {X 0,Y 278.471,Z 320.327,A -85,B 0,C 180,E1 -17327.045,E2 -17327.045} C_VEL
LIN {X 0,Y 278.358,Z 322.318,A -85,B 0,C 180,E1 -17329.239,E2 -17329.239} C_VEL
LIN {X 0,Y 278.11,Z 324.35,A -85,B 0,C 180,E1 -17331.404,E2 -17331.404} C_VEL
LIN {X 0,Y 279.133,Z 327.531,A -85,B 0,C 180,E1 -17331.707,E2 -17331.707} C_VEL
LIN {X 0,Y 280.861,Z 331.277,A -85,B 0,C 180,E1 -17332.125,E2 -17332.125} C_VEL
LIN {X 0,Y 286.208,Z 344.54,A -85,B 0,C 180,E1 -17333.606,E2 -17333.606} C_VEL
LIN {X 0,Y 289.829,Z 355.758,A -85,B 0,C 180,E1 -17334.864,E2 -17334.864} C_VEL
LIN {X 0,Y 292.796,Z 367.389,A -85,B 0,C 180,E1 -17336.231,E2 -17336.231} C_VEL
LIN {X 0,Y 295.267,Z 380.897,A -85,B 0,C 180,E1 -17337.904,E2 -17337.904} C_VEL
LIN {X 0,Y 296.199,Z 388.911,A -85,B 0,C 180,E1 -17338.96,E2 -17338.96} C_VEL
LIN {X 0,Y 293.633,Z 401.67,A -85,B 0,C 180,E1 -17340.419,E2 -17340.419} C_VEL
LIN {X 0,Y 290.789,Z 413.661,A -85,B 0,C 180,E1 -17342.078,E2 -17342.078} C_VEL
LIN {X 0,Y 287.999,Z 424.767,A -85,B 0,C 180,E1 -17343.944,E2 -17343.944} C_VEL
LIN {X 0,Y 285.134,Z 435.656,A -85,B 0,C 180,E1 -17346.17,E2 -17346.17} C_VEL
LIN {X 0,Y 282.537,Z 444.974,A -85,B 0,C 180,E1 -17348.475,E2 -17348.475} C_VEL
LIN {X 0,Y 280.321,Z 453.268,A -85,B 0,C 180,E1 -17350.978,E2 -17350.978} C_VEL
LIN {X 0,Y 278.28,Z 461.057,A -85,B 0,C 180,E1 -17353.87,E2 -17353.87} C_VEL
LIN {X 0,Y 276.892,Z 467.255,A -85,B 0,C 180,E1 -17356.795,E2 -17356.795} C_VEL
LIN {X 0,Y 275.917,Z 472.047,A -85,B 0,C 180,E1 -17359.729,E2 -17359.729} C_VEL
LIN {X 0,Y 275.414,Z 475.558,A -85,B 0,C 180,E1 -17362.669,E2 -17362.669} C_VEL
LIN {X 0,Y 275.2,Z 477.867,A -85,B 0,C 180,E1 -17365.606,E2 -17365.606} C_VEL
LIN {X 0,Y 275.219,Z 479.028,A -85,B 0,C 180,E1 -17368.536,E2 -17368.536} C_VEL
LIN {X 0,Y 275.219,Z 479.025,A -85,B 0,C 180,E1 -17371.463,E2 -17371.463} C_VEL
LIN {X 0,Y 275.202,Z 477.85,A -85,B 0,C 180,E1 -17374.393,E2 -17374.393} C_VEL
LIN {X 0,Y 275.414,Z 475.53,A -85,B 0,C 180,E1 -17377.33,E2 -17377.33} C_VEL
LIN {X 0,Y 275.916,Z 472.013,A -85,B 0,C 180,E1 -17380.27,E2 -17380.27} C_VEL
LIN {X 0,Y 276.89,Z 467.211,A -85,B 0,C 180,E1 -17383.204,E2 -17383.204} C_VEL
LIN {X 0,Y 278.298,Z 460.993,A -85,B 0,C 180,E1 -17386.127,E2 -17386.127} C_VEL
LIN {X 0,Y 280.312,Z 453.185,A -85,B 0,C 180,E1 -17389.021,E2 -17389.021} C_VEL
LIN {X 0,Y 282.536,Z 444.88,A -85,B 0,C 180,E1 -17391.524,E2 -17391.524} C_VEL
LIN {X 0,Y 285.225,Z 435.369,A -85,B 0,C 180,E1 -17393.867,E2 -17393.867} C_VEL
LIN {X 0,Y 287.982,Z 424.641,A -85,B 0,C 180,E1 -17396.057,E2 -17396.057} C_VEL
LIN {X 0,Y 291.048,Z 412.442,A -85,B 0,C 180,E1 -17398.09,E2 -17398.09} C_VEL
LIN {X 0,Y 294.22,Z 398.855,A -85,B 0,C 180,E1 -17399.909,E2 -17399.909} C_VEL
LIN {X 0,Y 296.048,Z 390.18,A -85,B 0,C 180,E1 -17400.868,E2 -17400.868} C_VEL
LIN {X 0,Y 295.511,Z 383.464,A -85,B 0,C 180,E1 -17401.744,E2 -17401.744} C_VEL
LIN {X 0,Y 293.233,Z 369.896,A -85,B 0,C 180,E1 -17403.451,E2 -17403.451} C_VEL
LIN {X 0,Y 290.286,Z 357.542,A -85,B 0,C 180,E1 -17404.902,E2 -17404.902} C_VEL
LIN {X 0,Y 286.39,Z 345.196,A -85,B 0,C 180,E1 -17406.291,E2 -17406.291} C_VEL
LIN {X 0,Y 281.278,Z 332.21,A -85,B 0,C 180,E1 -17407.733,E2 -17407.733} C_VEL
LIN {X 0,Y 279.241,Z 327.865,A -85,B 0,C 180,E1 -17408.221,E2 -17408.221} C_VEL
LIN {X 0,Y 278.168,Z 325.087,A -85,B 0,C 180,E1 -17408.498,E2 -17408.498} C_VEL
LIN {X 0,Y 278.073,Z 324.341,A -85,B 0,C 180,E1 -17408.581,E2 -17408.581} C_VEL
LIN {X 0,Y 278.375,Z 322.048,A -85,B 0,C 180,E1 -17411.025,E2 -17411.025} C_VEL
LIN {X 0,Y 278.484,Z 319.439,A -85,B 0,C 180,E1 -17413.946,E2 -17413.946} C_VEL
LIN {X 0,Y 278.2,Z 316.837,A -85,B 0,C 180,E1 -17417.104,E2 -17417.104} C_VEL
LIN {X 0,Y 277.749,Z 314.033,A -85,B 0,C 180,E1 -17420.759,E2 -17420.759} C_VEL
LIN {X 0,Y 277.385,Z 311.466,A -85,B 0,C 180,E1 -17424.357,E2 -17424.357} C_VEL
LIN {X 0,Y 277.241,Z 310.583,A -85,B 0,C 180,E1 -17426.104,E2 -17426.104} C_VEL
LIN {X 0,Y 277.256,Z 310.582,A -85,B 0,C 180,E1 -17429.538,E2 -17429.538} C_VEL
LIN {X 0,Y 277.352,Z 310.565,A -85,B 0,C 180,E1 -17432.864,E2 -17432.864} C_VEL
LIN {X 0,Y 277.322,Z 310.566,A -85,B 0,C 180,E1 -17436.079,E2 -17436.079} C_VEL
LIN {X 0,Y 277.339,Z 310.563,A -85,B 0,C 180,E1 -17440.766,E2 -17440.766} C_VEL
LIN {X 0,Y 277.422,Z 310.55,A -85,B 0,C 180,E1 -17445.325,E2 -17445.325} C_VEL
LIN {X 0,Y 277.451,Z 310.55,A -85,B 0,C 180,E1 -17449.787,E2 -17449.787} C_VEL
LIN {X 0,Y 277.594,Z 310.533,A -85,B 0,C 180,E1 -17452.728,E2 -17452.728} C_VEL
LIN {X 0,Y 277.692,Z 310.515,A -85,B 0,C 180,E1 -17457.099,E2 -17457.099} C_VEL
LIN {X 0,Y 277.855,Z 310.5,A -85,B 0,C 180,E1 -17460,E2 -17460} C_VEL
LIN {X 0,Y 277.692,Z 310.521,A -85,B 0,C 180,E1 -17462.902,E2 -17462.902} C_VEL
LIN {X 0,Y 277.594,Z 310.532,A -85,B 0,C 180,E1 -17467.273,E2 -17467.273} C_VEL
LIN {X 0,Y 277.451,Z 310.551,A -85,B 0,C 180,E1 -17470.214,E2 -17470.214} C_VEL
LIN {X 0,Y 277.422,Z 310.549,A -85,B 0,C 180,E1 -17474.675,E2 -17474.675} C_VEL
LIN {X 0,Y 277.339,Z 310.564,A -85,B 0,C 180,E1 -17479.234,E2 -17479.234} C_VEL
LIN {X 0,Y 277.314,Z 310.568,A -85,B 0,C 180,E1 -17484.171,E2 -17484.171} C_VEL
LIN {X 0,Y 277.318,Z 310.565,A -85,B 0,C 180,E1 -17487.505,E2 -17487.505} C_VEL
LIN {X 0,Y 277.267,Z 310.569,A -85,B 0,C 180,E1 -17490.482,E2 -17490.482} C_VEL
LIN {X 0,Y 277.242,Z 310.572,A -85,B 0,C 180,E1 -17493.897,E2 -17493.897} C_VEL
LIN {X 0,Y 277.263,Z 310.572,A -85,B 0,C 180,E1 -17497.47,E2 -17497.47} C_VEL
LIN {X 0,Y 277.286,Z 310.703,A -85,B 0,C 180,E1 -17498.215,E2 -17498.215} C_VEL
LIN {X 0,Y 277.557,Z 312.643,A -85,B 0,C 180,E1 -17501.174,E2 -17501.174} C_VEL
LIN {X 0,Y 277.948,Z 315.373,A -85,B 0,C 180,E1 -17505.072,E2 -17505.072} C_VEL
LIN {X 0,Y 277.999,Z 316.95,A -85,B 0,C 180,E1 -17507.15,E2 -17507.15} C_VEL
LIN {X 0,Y 277.783,Z 319.845,A -85,B 0,C 180,E1 -17510.766,E2 -17510.766} C_VEL
LIN {X 0,Y 277.757,Z 320.594,A -85,B 0,C 180,E1 -17511.471,E2 -17511.471} C_VEL
LIN {X 0,Y 278.843,Z 323.688,A -85,B 0,C 180,E1 -17511.763,E2 -17511.763} C_VEL
LIN {X 0,Y 280.107,Z 326.123,A -85,B 0,C 180,E1 -17512.059,E2 -17512.059} C_VEL
LIN {X 0,Y 285.246,Z 337.877,A -85,B 0,C 180,E1 -17513.414,E2 -17513.414} C_VEL
LIN {X 0,Y 289.377,Z 349.278,A -85,B 0,C 180,E1 -17514.749,E2 -17514.749} C_VEL
LIN {X 0,Y 292.912,Z 361.421,A -85,B 0,C 180,E1 -17516.211,E2 -17516.211} C_VEL
LIN {X 0,Y 295.838,Z 375.43,A -85,B 0,C 180,E1 -17517.982,E2 -17517.982} C_VEL
LIN {X 0,Y 296.743,Z 383.441,A -85,B 0,C 180,E1 -17519.033,E2 -17519.033} C_VEL
LIN {X 0,Y 294.064,Z 396.224,A -85,B 0,C 180,E1 -17520.468,E2 -17520.468} C_VEL
LIN {X 0,Y 291.335,Z 408.267,A -85,B 0,C 180,E1 -17522.136,E2 -17522.136} C_VEL
LIN {X 0,Y 288.521,Z 419.397,A -85,B 0,C 180,E1 -17523.996,E2 -17523.996} C_VEL
LIN {X 0,Y 285.859,Z 429.61,A -85,B 0,C 180,E1 -17526.068,E2 -17526.068} C_VEL
LIN {X 0,Y 283.071,Z 439.605,A -85,B 0,C 180,E1 -17528.519,E2 -17528.519} C_VEL
LIN {X 0,Y 280.767,Z 447.895,A -85,B 0,C 180,E1 -17531.011,E2 -17531.011} C_VEL
LIN {X 0,Y 278.707,Z 455.682,A -85,B 0,C 180,E1 -17533.897,E2 -17533.897} C_VEL
LIN {X 0,Y 277.167,Z 461.881,A -85,B 0,C 180,E1 -17536.809,E2 -17536.809} C_VEL
LIN {X 0,Y 276.169,Z 466.667,A -85,B 0,C 180,E1 -17539.739,E2 -17539.739} C_VEL
LIN {X 0,Y 275.526,Z 470.173,A -85,B 0,C 180,E1 -17542.673,E2 -17542.673} C_VEL
LIN {X 0,Y 275.274,Z 472.489,A -85,B 0,C 180,E1 -17545.608,E2 -17545.608} C_VEL
LIN {X 0,Y 275.234,Z 473.67,A -85,B 0,C 180,E1 -17548.537,E2 -17548.537} C_VEL
LIN {X 0,Y 275.234,Z 473.683,A -85,B 0,C 180,E1 -17551.464,E2 -17551.464} C_VEL
LIN {X 0,Y 275.274,Z 472.555,A -85,B 0,C 180,E1 -17554.393,E2 -17554.393} C_VEL
LIN {X 0,Y 275.526,Z 470.29,A -85,B 0,C 180,E1 -17557.328,E2 -17557.328} C_VEL
LIN {X 0,Y 276.147,Z 466.83,A -85,B 0,C 180,E1 -17560.263,E2 -17560.263} C_VEL
LIN {X 0,Y 277.147,Z 462.096,A -85,B 0,C 180,E1 -17563.193,E2 -17563.193} C_VEL
LIN {X 0,Y 278.643,Z 455.963,A -85,B 0,C 180,E1 -17566.108,E2 -17566.108} C_VEL
LIN {X 0,Y 280.673,Z 448.243,A -85,B 0,C 180,E1 -17568.997,E2 -17568.997} C_VEL
LIN {X 0,Y 282.986,Z 440.013,A -85,B 0,C 180,E1 -17571.489,E2 -17571.489} C_VEL
LIN {X 0,Y 285.79,Z 430.098,A -85,B 0,C 180,E1 -17573.939,E2 -17573.939} C_VEL
LIN {X 0,Y 288.422,Z 419.938,A -85,B 0,C 180,E1 -17576.015,E2 -17576.015} C_VEL
LIN {X 0,Y 291.222,Z 408.906,A -85,B 0,C 180,E1 -17577.877,E2 -17577.877} C_VEL
LIN {X 0,Y 293.931,Z 396.996,A -85,B 0,C 180,E1 -17579.548,E2 -17579.548} C_VEL
LIN {X 0,Y 296.736,Z 384,A -85,B 0,C 180,E1 -17581.019,E2 -17581.019} C_VEL
LIN {X 0,Y 296.416,Z 379.353,A -85,B 0,C 180,E1 -17581.624,E2 -17581.624} C_VEL
LIN {X 0,Y 294.17,Z 366.728,A -85,B 0,C 180,E1 -17583.261,E2 -17583.261} C_VEL
LIN {X 0,Y 290.521,Z 352.671,A -85,B 0,C 180,E1 -17584.968,E2 -17584.968} C_VEL
LIN {X 0,Y 285.94,Z 339.451,A -85,B 0,C 180,E1 -17586.515,E2 -17586.515} C_VEL
LIN {X 0,Y 280.965,Z 327.956,A -85,B 0,C 180,E1 -17587.866,E2 -17587.866} C_VEL
LIN {X 0,Y 279.121,Z 324.159,A -85,B 0,C 180,E1 -17588.306,E2 -17588.306} C_VEL
LIN {X 0,Y 277.869,Z 321.248,A -85,B 0,C 180,E1 -17588.622,E2 -17588.622} C_VEL
LIN {X 0,Y 277.732,Z 320.4,A -85,B 0,C 180,E1 -17588.714,E2 -17588.714} C_VEL
LIN {X 0,Y 277.949,Z 318.433,A -85,B 0,C 180,E1 -17591.103,E2 -17591.103} C_VEL
LIN {X 0,Y 278.012,Z 316.914,A -85,B 0,C 180,E1 -17593.043,E2 -17593.043} C_VEL
LIN {X 0,Y 277.947,Z 315.381,A -85,B 0,C 180,E1 -17595.071,E2 -17595.071} C_VEL
LIN {X 0,Y 277.513,Z 312.334,A -85,B 0,C 180,E1 -17599.442,E2 -17599.442} C_VEL
LIN {X 0,Y 277.309,Z 310.807,A -85,B 0,C 180,E1 -17601.78,E2 -17601.78} C_VEL
LIN {X 0,Y 277.284,Z 310.574,A -85,B 0,C 180,E1 -17604.341,E2 -17604.341} C_VEL
LIN {X 0,Y 277.239,Z 310.577,A -85,B 0,C 180,E1 -17607.835,E2 -17607.835} C_VEL
LIN {X 0,Y 277.239,Z 310.575,A -85,B 0,C 180,E1 -17611.207,E2 -17611.207} C_VEL
LIN {X 0,Y 277.246,Z 310.576,A -85,B 0,C 180,E1 -17614.473,E2 -17614.473} C_VEL
LIN {X 0,Y 277.266,Z 310.57,A -85,B 0,C 180,E1 -17617.653,E2 -17617.653} C_VEL
LIN {X 0,Y 277.344,Z 310.559,A -85,B 0,C 180,E1 -17620.766,E2 -17620.766} C_VEL
LIN {X 0,Y 277.434,Z 310.553,A -85,B 0,C 180,E1 -17625.326,E2 -17625.326} C_VEL
LIN {X 0,Y 277.456,Z 310.549,A -85,B 0,C 180,E1 -17629.787,E2 -17629.787} C_VEL
LIN {X 0,Y 277.6,Z 310.532,A -85,B 0,C 180,E1 -17632.728,E2 -17632.728} C_VEL
LIN {X 0,Y 277.696,Z 310.519,A -85,B 0,C 180,E1 -17637.098,E2 -17637.098} C_VEL
LIN {X 0,Y 277.851,Z 310.501,A -85,B 0,C 180,E1 -17640,E2 -17640} C_VEL
LIN {X 0,Y 277.746,Z 310.51,A -85,B 0,C 180,E1 -17642.038,E2 -17642.038} C_VEL
LIN {X 0,Y 276.993,Z 310.608,A -85,B 0,C 180,E1 -17643.246,E2 -17643.246} C_VEL
LIN {X 0,Y 274.068,Z 310.971,A -85,B 0,C 180,E1 -17645.214,E2 -17645.214} C_VEL
LIN {X 0,Y 271.634,Z 311.273,A -85,B 0,C 180,E1 -17646.813,E2 -17646.813} C_VEL
LIN {X 0,Y 270.599,Z 311.404,A -85,B 0,C 180,E1 -17648.054,E2 -17648.054} C_VEL
LIN {X 0,Y 270.517,Z 311.411,A -85,B 0,C 180,E1 -17648.474,E2 -17648.474} C_VEL
LIN {X 0,Y 270.394,Z 311.431,A -85,B 0,C 180,E1 -17652.001,E2 -17652.001} C_VEL
LIN {X 0,Y 270.38,Z 311.431,A -85,B 0,C 180,E1 -17655.901,E2 -17655.901} C_VEL
LIN {X 0,Y 270.29,Z 311.442,A -85,B 0,C 180,E1 -17660.601,E2 -17660.601} C_VEL
LIN {X 0,Y 270.237,Z 311.45,A -85,B 0,C 180,E1 -17664.589,E2 -17664.589} C_VEL
LIN {X 0,Y 270.269,Z 311.447,A -85,B 0,C 180,E1 -17667.909,E2 -17667.909} C_VEL
LIN {X 0,Y 270.183,Z 311.463,A -85,B 0,C 180,E1 -17671.348,E2 -17671.348} C_VEL
LIN {X 0,Y 270.215,Z 311.56,A -85,B 0,C 180,E1 -17673.666,E2 -17673.666} C_VEL
LIN {X 0,Y 270.503,Z 313.538,A -85,B 0,C 180,E1 -17676.696,E2 -17676.696} C_VEL
LIN {X 0,Y 270.918,Z 316.187,A -85,B 0,C 180,E1 -17680.431,E2 -17680.431} C_VEL
LIN {X 0,Y 271.327,Z 319.229,A -85,B 0,C 180,E1 -17684.376,E2 -17684.376} C_VEL
LIN {X 0,Y 271.476,Z 320.934,A -85,B 0,C 180,E1 -17686.458,E2 -17686.458} C_VEL
LIN {X 0,Y 271.228,Z 324.388,A -85,B 0,C 180,E1 -17690.261,E2 -17690.261} C_VEL
LIN {X 0,Y 272.176,Z 327.356,A -85,B 0,C 180,E1 -17690.537,E2 -17690.537} C_VEL
LIN {X 0,Y 273.422,Z 329.741,A -85,B 0,C 180,E1 -17690.845,E2 -17690.845} C_VEL
LIN {X 0,Y 278.4,Z 341.503,A -85,B 0,C 180,E1 -17692.228,E2 -17692.228} C_VEL
LIN {X 0,Y 282.692,Z 353.901,A -85,B 0,C 180,E1 -17693.71,E2 -17693.71} C_VEL
LIN {X 0,Y 286.238,Z 367.221,A -85,B 0,C 180,E1 -17695.339,E2 -17695.339} C_VEL
LIN {X 0,Y 288.756,Z 381.098,A -85,B 0,C 180,E1 -17697.121,E2 -17697.121} C_VEL
LIN {X 0,Y 289.804,Z 390.137,A -85,B 0,C 180,E1 -17698.362,E2 -17698.362} C_VEL
LIN {X 0,Y 288.08,Z 398.99,A -85,B 0,C 180,E1 -17699.385,E2 -17699.385} C_VEL
LIN {X 0,Y 284.795,Z 412.524,A -85,B 0,C 180,E1 -17701.235,E2 -17701.235} C_VEL
LIN {X 0,Y 281.608,Z 424.701,A -85,B 0,C 180,E1 -17703.306,E2 -17703.306} C_VEL
LIN {X 0,Y 278.891,Z 434.221,A -85,B 0,C 180,E1 -17705.26,E2 -17705.26} C_VEL
LIN {X 0,Y 276.319,Z 443.552,A -85,B 0,C 180,E1 -17707.572,E2 -17707.572} C_VEL
LIN {X 0,Y 273.853,Z 452.081,A -85,B 0,C 180,E1 -17710.12,E2 -17710.12} C_VEL
LIN {X 0,Y 271.87,Z 459.178,A -85,B 0,C 180,E1 -17712.706,E2 -17712.706} C_VEL
LIN {X 0,Y 270.272,Z 465.759,A -85,B 0,C 180,E1 -17715.698,E2 -17715.698} C_VEL
LIN {X 0,Y 269.07,Z 470.908,A -85,B 0,C 180,E1 -17718.702,E2 -17718.702} C_VEL
LIN {X 0,Y 268.583,Z 473.889,A -85,B 0,C 180,E1 -17720.967,E2 -17720.967} C_VEL
LIN {X 0,Y 268.208,Z 476.79,A -85,B 0,C 180,E1 -17723.983,E2 -17723.983} C_VEL
LIN {X 0,Y 268.099,Z 478.52,A -85,B 0,C 180,E1 -17726.994,E2 -17726.994} C_VEL
LIN {X 0,Y 268.143,Z 479.112,A -85,B 0,C 180,E1 -17729.999,E2 -17729.999} C_VEL
LIN {X 0,Y 268.1,Z 478.51,A -85,B 0,C 180,E1 -17733.005,E2 -17733.005} C_VEL
LIN {X 0,Y 268.207,Z 476.766,A -85,B 0,C 180,E1 -17736.016,E2 -17736.016} C_VEL
LIN {X 0,Y 268.582,Z 473.856,A -85,B 0,C 180,E1 -17739.032,E2 -17739.032} C_VEL
LIN {X 0,Y 269.289,Z 469.709,A -85,B 0,C 180,E1 -17742.05,E2 -17742.05} C_VEL
LIN {X 0,Y 270.599,Z 464.218,A -85,B 0,C 180,E1 -17745.053,E2 -17745.053} C_VEL
LIN {X 0,Y 272.349,Z 457.23,A -85,B 0,C 180,E1 -17748.038,E2 -17748.038} C_VEL
LIN {X 0,Y 274.491,Z 449.755,A -85,B 0,C 180,E1 -17750.612,E2 -17750.612} C_VEL
LIN {X 0,Y 277.189,Z 440.743,A -85,B 0,C 180,E1 -17753.14,E2 -17753.14} C_VEL
LIN {X 0,Y 280.153,Z 429.908,A -85,B 0,C 180,E1 -17755.64,E2 -17755.64} C_VEL
LIN {X 0,Y 283.149,Z 418.749,A -85,B 0,C 180,E1 -17757.734,E2 -17757.734} C_VEL
LIN {X 0,Y 286.236,Z 406.519,A -85,B 0,C 180,E1 -17759.611,E2 -17759.611} C_VEL
LIN {X 0,Y 289.443,Z 392.693,A -85,B 0,C 180,E1 -17761.317,E2 -17761.317} C_VEL
LIN {X 0,Y 289.695,Z 389.95,A -85,B 0,C 180,E1 -17761.642,E2 -17761.642} C_VEL
LIN {X 0,Y 288.006,Z 376.676,A -85,B 0,C 180,E1 -17763.437,E2 -17763.437} C_VEL
LIN {X 0,Y 285.11,Z 362.882,A -85,B 0,C 180,E1 -17765.182,E2 -17765.182} C_VEL
LIN {X 0,Y 281.3,Z 349.639,A -85,B 0,C 180,E1 -17766.77,E2 -17766.77} C_VEL
LIN {X 0,Y 276.134,Z 335.972,A -85,B 0,C 180,E1 -17768.381,E2 -17768.381} C_VEL
LIN {X 0,Y 272.457,Z 327.93,A -85,B 0,C 180,E1 -17769.347,E2 -17769.347} C_VEL
LIN {X 0,Y 271.287,Z 324.996,A -85,B 0,C 180,E1 -17769.662,E2 -17769.662} C_VEL
LIN {X 0,Y 271.167,Z 324.288,A -85,B 0,C 180,E1 -17769.726,E2 -17769.726} C_VEL
LIN {X 0,Y 271.393,Z 321.959,A -85,B 0,C 180,E1 -17772.32,E2 -17772.32} C_VEL
LIN {X 0,Y 271.458,Z 320.231,A -85,B 0,C 180,E1 -17774.347,E2 -17774.347} C_VEL
LIN {X 0,Y 271.112,Z 317.63,A -85,B 0,C 180,E1 -17777.624,E2 -17777.624} C_VEL
LIN {X 0,Y 270.704,Z 314.789,A -85,B 0,C 180,E1 -17781.458,E2 -17781.458} C_VEL
LIN {X 0,Y 270.297,Z 312.299,A -85,B 0,C 180,E1 -17785.109,E2 -17785.109} C_VEL
LIN {X 0,Y 270.21,Z 311.51,A -85,B 0,C 180,E1 -17786.333,E2 -17786.333} C_VEL
LIN {X 0,Y 270.19,Z 311.462,A -85,B 0,C 180,E1 -17790.382,E2 -17790.382} C_VEL
LIN {X 0,Y 270.257,Z 311.451,A -85,B 0,C 180,E1 -17793.763,E2 -17793.763} C_VEL
LIN {X 0,Y 270.227,Z 311.451,A -85,B 0,C 180,E1 -17797.038,E2 -17797.038} C_VEL
LIN {X 0,Y 270.296,Z 311.439,A -85,B 0,C 180,E1 -17800.244,E2 -17800.244} C_VEL
LIN {X 0,Y 270.39,Z 311.426,A -85,B 0,C 180,E1 -17804.935,E2 -17804.935} C_VEL
LIN {X 0,Y 270.403,Z 311.429,A -85,B 0,C 180,E1 -17809.518,E2 -17809.518} C_VEL
LIN {X 0,Y 270.556,Z 311.41,A -85,B 0,C 180,E1 -17812.537,E2 -17812.537} C_VEL
LIN {X 0,Y 270.779,Z 311.378,A -85,B 0,C 180,E1 -17818.513,E2 -17818.513} C_VEL
LIN {X 0,Y 270.779,Z 311.382,A -85,B 0,C 180,E1 -17821.487,E2 -17821.487} C_VEL
LIN {X 0,Y 270.556,Z 311.406,A -85,B 0,C 180,E1 -17827.463,E2 -17827.463} C_VEL
LIN {X 0,Y 270.404,Z 311.428,A -85,B 0,C 180,E1 -17830.483,E2 -17830.483} C_VEL
LIN {X 0,Y 270.391,Z 311.425,A -85,B 0,C 180,E1 -17835.066,E2 -17835.066} C_VEL
LIN {X 0,Y 270.296,Z 311.44,A -85,B 0,C 180,E1 -17839.756,E2 -17839.756} C_VEL
LIN {X 0,Y 270.269,Z 311.444,A -85,B 0,C 180,E1 -17844.586,E2 -17844.586} C_VEL
LIN {X 0,Y 270.265,Z 311.441,A -85,B 0,C 180,E1 -17847.91,E2 -17847.91} C_VEL
LIN {X 0,Y 270.179,Z 311.451,A -85,B 0,C 180,E1 -17851.349,E2 -17851.349} C_VEL
LIN {X 0,Y 270.197,Z 311.45,A -85,B 0,C 180,E1 -17854.906,E2 -17854.906} C_VEL
LIN {X 0,Y 270.213,Z 311.45,A -85,B 0,C 180,E1 -17856.742,E2 -17856.742} C_VEL
LIN {X 0,Y 270.33,Z 312.308,A -85,B 0,C 180,E1 -17858.747,E2 -17858.747} C_VEL
LIN {X 0,Y 270.652,Z 314.736,A -85,B 0,C 180,E1 -17862.465,E2 -17862.465} C_VEL
LIN {X 0,Y 270.932,Z 316.872,A -85,B 0,C 180,E1 -17865.544,E2 -17865.544} C_VEL
LIN {X 0,Y 270.934,Z 319.323,A -85,B 0,C 180,E1 -17868.787,E2 -17868.787} C_VEL
LIN {X 0,Y 270.796,Z 320.553,A -85,B 0,C 180,E1 -17870.283,E2 -17870.283} C_VEL
LIN {X 0,Y 271.865,Z 323.675,A -85,B 0,C 180,E1 -17870.589,E2 -17870.589} C_VEL
LIN {X 0,Y 273.075,Z 325.719,A -85,B 0,C 180,E1 -17870.879,E2 -17870.879} C_VEL
LIN {X 0,Y 279.112,Z 339.358,A -85,B 0,C 180,E1 -17872.56,E2 -17872.56} C_VEL
LIN {X 0,Y 283.451,Z 351.575,A -85,B 0,C 180,E1 -17874.058,E2 -17874.058} C_VEL
LIN {X 0,Y 286.708,Z 363.104,A -85,B 0,C 180,E1 -17875.529,E2 -17875.529} C_VEL
LIN {X 0,Y 289.319,Z 375.793,A -85,B 0,C 180,E1 -17877.205,E2 -17877.205} C_VEL
LIN {X 0,Y 290.419,Z 384.687,A -85,B 0,C 180,E1 -17878.432,E2 -17878.432} C_VEL
LIN {X 0,Y 287.587,Z 397.587,A -85,B 0,C 180,E1 -17879.937,E2 -17879.937} C_VEL
LIN {X 0,Y 284.777,Z 409.407,A -85,B 0,C 180,E1 -17881.637,E2 -17881.637} C_VEL
LIN {X 0,Y 281.833,Z 420.549,A -85,B 0,C 180,E1 -17883.573,E2 -17883.573} C_VEL
LIN {X 0,Y 278.933,Z 431.212,A -85,B 0,C 180,E1 -17885.832,E2 -17885.832} C_VEL
LIN {X 0,Y 276.426,Z 439.677,A -85,B 0,C 180,E1 -17887.976,E2 -17887.976} C_VEL
LIN {X 0,Y 274.01,Z 447.966,A -85,B 0,C 180,E1 -17890.524,E2 -17890.524} C_VEL
LIN {X 0,Y 271.851,Z 455.753,A -85,B 0,C 180,E1 -17893.479,E2 -17893.479} C_VEL
LIN {X 0,Y 270.237,Z 461.951,A -85,B 0,C 180,E1 -17896.465,E2 -17896.465} C_VEL
LIN {X 0,Y 269.164,Z 466.737,A -85,B 0,C 180,E1 -17899.469,E2 -17899.469} C_VEL
LIN {X 0,Y 268.478,Z 470.243,A -85,B 0,C 180,E1 -17902.48,E2 -17902.48} C_VEL
LIN {X 0,Y 268.191,Z 472.559,A -85,B 0,C 180,E1 -17905.492,E2 -17905.492} C_VEL
LIN {X 0,Y 268.14,Z 473.739,A -85,B 0,C 180,E1 -17908.499,E2 -17908.499} C_VEL
LIN {X 0,Y 268.141,Z 473.752,A -85,B 0,C 180,E1 -17911.502,E2 -17911.502} C_VEL
LIN {X 0,Y 268.191,Z 472.624,A -85,B 0,C 180,E1 -17914.509,E2 -17914.509} C_VEL
LIN {X 0,Y 268.478,Z 470.358,A -85,B 0,C 180,E1 -17917.521,E2 -17917.521} C_VEL
LIN {X 0,Y 269.14,Z 466.899,A -85,B 0,C 180,E1 -17920.533,E2 -17920.533} C_VEL
LIN {X 0,Y 270.217,Z 462.164,A -85,B 0,C 180,E1 -17923.538,E2 -17923.538} C_VEL
LIN {X 0,Y 271.782,Z 456.031,A -85,B 0,C 180,E1 -17926.526,E2 -17926.526} C_VEL
LIN {X 0,Y 273.938,Z 448.31,A -85,B 0,C 180,E1 -17929.483,E2 -17929.483} C_VEL
LIN {X 0,Y 276.316,Z 440.08,A -85,B 0,C 180,E1 -17932.034,E2 -17932.034} C_VEL
LIN {X 0,Y 279.28,Z 430.165,A -85,B 0,C 180,E1 -17934.533,E2 -17934.533} C_VEL
LIN {X 0,Y 282.027,Z 420.004,A -85,B 0,C 180,E1 -17936.651,E2 -17936.651} C_VEL
LIN {X 0,Y 285.211,Z 407.904,A -85,B 0,C 180,E1 -17938.719,E2 -17938.719} C_VEL
LIN {X 0,Y 288.093,Z 395.771,A -85,B 0,C 180,E1 -17940.411,E2 -17940.411} C_VEL
LIN {X 0,Y 290.415,Z 385.293,A -85,B 0,C 180,E1 -17941.613,E2 -17941.613} C_VEL
LIN {X 0,Y 289.792,Z 378.49,A -85,B 0,C 180,E1 -17942.543,E2 -17942.543} C_VEL
LIN {X 0,Y 287.44,Z 366.041,A -85,B 0,C 180,E1 -17944.219,E2 -17944.219} C_VEL
LIN {X 0,Y 283.99,Z 353.18,A -85,B 0,C 180,E1 -17945.858,E2 -17945.858} C_VEL
LIN {X 0,Y 279.202,Z 339.501,A -85,B 0,C 180,E1 -17947.547,E2 -17947.547} C_VEL
LIN {X 0,Y 274.068,Z 327.982,A -85,B 0,C 180,E1 -17948.997,E2 -17948.997} C_VEL
LIN {X 0,Y 272.359,Z 324.398,A -85,B 0,C 180,E1 -17949.432,E2 -17949.432} C_VEL
LIN {X 0,Y 271.027,Z 321.623,A -85,B 0,C 180,E1 -17949.775,E2 -17949.775} C_VEL
LIN {X 0,Y 270.811,Z 320.482,A -85,B 0,C 180,E1 -17949.891,E2 -17949.891} C_VEL
LIN {X 0,Y 270.992,Z 317.735,A -85,B 0,C 180,E1 -17953.434,E2 -17953.434} C_VEL
LIN {X 0,Y 270.767,Z 315.459,A -85,B 0,C 180,E1 -17956.616,E2 -17956.616} C_VEL
LIN {X 0,Y 270.53,Z 313.526,A -85,B 0,C 180,E1 -17959.498,E2 -17959.498} C_VEL
LIN {X 0,Y 270.217,Z 311.454,A -85,B 0,C 180,E1 -17963.259,E2 -17963.259} C_VEL
LIN {X 0,Y 270.201,Z 311.456,A -85,B 0,C 180,E1 -17966.892,E2 -17966.892} C_VEL
LIN {X 0,Y 270.182,Z 311.457,A -85,B 0,C 180,E1 -17970.381,E2 -17970.381} C_VEL
LIN {X 0,Y 270.202,Z 311.452,A -85,B 0,C 180,E1 -17973.757,E2 -17973.757} C_VEL
LIN {X 0,Y 270.203,Z 311.453,A -85,B 0,C 180,E1 -17977.036,E2 -17977.036} C_VEL
LIN {X 0,Y 270.301,Z 311.437,A -85,B 0,C 180,E1 -17980.244,E2 -17980.244} C_VEL
LIN {X 0,Y 270.402,Z 311.428,A -85,B 0,C 180,E1 -17984.935,E2 -17984.935} C_VEL
LIN {X 0,Y 270.409,Z 311.427,A -85,B 0,C 180,E1 -17989.518,E2 -17989.518} C_VEL
LIN {X 0,Y 270.561,Z 311.41,A -85,B 0,C 180,E1 -17992.537,E2 -17992.537} C_VEL
LIN {X 0,Y 270.784,Z 311.382,A -85,B 0,C 180,E1 -17998.513,E2 -17998.513} C_VEL
LIN {X 0,Y 270.709,Z 311.387,A -85,B 0,C 180,E1 -18001.999,E2 -18001.999} C_VEL
LIN {X 0,Y 270.561,Z 311.408,A -85,B 0,C 180,E1 -18007.462,E2 -18007.462} C_VEL
LIN {X 0,Y 270.517,Z 311.411,A -85,B 0,C 180,E1 -18008.474,E2 -18008.474} C_VEL
LIN {X 0,Y 269.828,Z 311.501,A -85,B 0,C 180,E1 -18009.716,E2 -18009.716} C_VEL
LIN {X 0,Y 266.878,Z 311.868,A -85,B 0,C 180,E1 -18011.735,E2 -18011.735} C_VEL
LIN {X 0,Y 264.402,Z 312.177,A -85,B 0,C 180,E1 -18013.378,E2 -18013.378} C_VEL
LIN {X 0,Y 263.381,Z 312.303,A -85,B 0,C 180,E1 -18014.654,E2 -18014.654} C_VEL
LIN {X 0,Y 263.32,Z 312.309,A -85,B 0,C 180,E1 -18015.087,E2 -18015.087} C_VEL
LIN {X 0,Y 263.247,Z 312.32,A -85,B 0,C 180,E1 -18018.685,E2 -18018.685} C_VEL
LIN {X 0,Y 263.145,Z 312.332,A -85,B 0,C 180,E1 -18021.957,E2 -18021.957} C_VEL
LIN {X 0,Y 263.191,Z 312.326,A -85,B 0,C 180,E1 -18025.293,E2 -18025.293} C_VEL
LIN {X 0,Y 263.165,Z 312.335,A -85,B 0,C 180,E1 -18028.731,E2 -18028.731} C_VEL
LIN {X 0,Y 263.132,Z 312.343,A -85,B 0,C 180,E1 -18032.288,E2 -18032.288} C_VEL
LIN {X 0,Y 263.455,Z 314.345,A -85,B 0,C 180,E1 -18035.936,E2 -18035.936} C_VEL
LIN {X 0,Y 263.846,Z 316.933,A -85,B 0,C 180,E1 -18039.738,E2 -18039.738} C_VEL
LIN {X 0,Y 264.273,Z 319.882,A -85,B 0,C 180,E1 -18043.744,E2 -18043.744} C_VEL
LIN {X 0,Y 264.468,Z 321.92,A -85,B 0,C 180,E1 -18046.297,E2 -18046.297} C_VEL
LIN {X 0,Y 264.299,Z 324.191,A -85,B 0,C 180,E1 -18048.978,E2 -18048.978} C_VEL
LIN {X 0,Y 265.353,Z 327.397,A -85,B 0,C 180,E1 -18049.317,E2 -18049.317} C_VEL
LIN {X 0,Y 266.605,Z 329.649,A -85,B 0,C 180,E1 -18049.64,E2 -18049.64} C_VEL
LIN {X 0,Y 271.702,Z 341.288,A -85,B 0,C 180,E1 -18051.116,E2 -18051.116} C_VEL
LIN {X 0,Y 276.699,Z 355.662,A -85,B 0,C 180,E1 -18052.93,E2 -18052.93} C_VEL
LIN {X 0,Y 280.356,Z 370.107,A -85,B 0,C 180,E1 -18054.79,E2 -18054.79} C_VEL
LIN {X 0,Y 282.595,Z 383.573,A -85,B 0,C 180,E1 -18056.617,E2 -18056.617} C_VEL
LIN {X 0,Y 283.43,Z 392.617,A -85,B 0,C 180,E1 -18057.905,E2 -18057.905} C_VEL
LIN {X 0,Y 280.397,Z 405.414,A -85,B 0,C 180,E1 -18059.499,E2 -18059.499} C_VEL
LIN {X 0,Y 277.089,Z 417.811,A -85,B 0,C 180,E1 -18061.397,E2 -18061.397} C_VEL
LIN {X 0,Y 273.68,Z 429.964,A -85,B 0,C 180,E1 -18063.706,E2 -18063.706} C_VEL
LIN {X 0,Y 271.004,Z 439.34,A -85,B 0,C 180,E1 -18065.892,E2 -18065.892} C_VEL
LIN {X 0,Y 268.177,Z 448.561,A -85,B 0,C 180,E1 -18068.476,E2 -18068.476} C_VEL
LIN {X 0,Y 265.561,Z 457.24,A -85,B 0,C 180,E1 -18071.483,E2 -18071.483} C_VEL
LIN {X 0,Y 263.683,Z 464.205,A -85,B 0,C 180,E1 -18074.542,E2 -18074.542} C_VEL
LIN {X 0,Y 262.299,Z 469.68,A -85,B 0,C 180,E1 -18077.622,E2 -18077.622} C_VEL
LIN {X 0,Y 261.525,Z 473.82,A -85,B 0,C 180,E1 -18080.721,E2 -18080.721} C_VEL
LIN {X 0,Y 261.136,Z 476.722,A -85,B 0,C 180,E1 -18083.819,E2 -18083.819} C_VEL
LIN {X 0,Y 260.998,Z 478.451,A -85,B 0,C 180,E1 -18086.912,E2 -18086.912} C_VEL
LIN {X 0,Y 261.071,Z 479.043,A -85,B 0,C 180,E1 -18089.999,E2 -18089.999} C_VEL
LIN {X 0,Y 260.998,Z 478.44,A -85,B 0,C 180,E1 -18093.086,E2 -18093.086} C_VEL
LIN {X 0,Y 261.135,Z 476.697,A -85,B 0,C 180,E1 -18096.179,E2 -18096.179} C_VEL
LIN {X 0,Y 261.524,Z 473.786,A -85,B 0,C 180,E1 -18099.278,E2 -18099.278} C_VEL
LIN {X 0,Y 262.297,Z 469.639,A -85,B 0,C 180,E1 -18102.377,E2 -18102.377} C_VEL
LIN {X 0,Y 263.689,Z 464.147,A -85,B 0,C 180,E1 -18105.457,E2 -18105.457} C_VEL
LIN {X 0,Y 265.558,Z 457.159,A -85,B 0,C 180,E1 -18108.516,E2 -18108.516} C_VEL
LIN {X 0,Y 268.132,Z 448.464,A -85,B 0,C 180,E1 -18111.527,E2 -18111.527} C_VEL
LIN {X 0,Y 271.034,Z 439.228,A -85,B 0,C 180,E1 -18114.104,E2 -18114.104} C_VEL
LIN {X 0,Y 273.717,Z 429.835,A -85,B 0,C 180,E1 -18116.289,E2 -18116.289} C_VEL
LIN {X 0,Y 276.853,Z 418.676,A -85,B 0,C 180,E1 -18118.422,E2 -18118.422} C_VEL
LIN {X 0,Y 280.071,Z 406.447,A -85,B 0,C 180,E1 -18120.331,E2 -18120.331} C_VEL
LIN {X 0,Y 283.398,Z 392.619,A -85,B 0,C 180,E1 -18122.064,E2 -18122.064} C_VEL
LIN {X 0,Y 282.119,Z 380.639,A -85,B 0,C 180,E1 -18123.764,E2 -18123.764} C_VEL
LIN {X 0,Y 279.775,Z 367.917,A -85,B 0,C 180,E1 -18125.468,E2 -18125.468} C_VEL
LIN {X 0,Y 276.087,Z 353.878,A -85,B 0,C 180,E1 -18127.259,E2 -18127.259} C_VEL
LIN {X 0,Y 270.954,Z 339.649,A -85,B 0,C 180,E1 -18129.057,E2 -18129.057} C_VEL
LIN {X 0,Y 267.472,Z 331.763,A -85,B 0,C 180,E1 -18130.068,E2 -18130.068} C_VEL
LIN {X 0,Y 265.742,Z 328.122,A -85,B 0,C 180,E1 -18130.532,E2 -18130.532} C_VEL
LIN {X 0,Y 264.4,Z 324.954,A -85,B 0,C 180,E1 -18130.909,E2 -18130.909} C_VEL
LIN {X 0,Y 264.311,Z 324.161,A -85,B 0,C 180,E1 -18131.019,E2 -18131.019} C_VEL
LIN {X 0,Y 264.472,Z 321.519,A -85,B 0,C 180,E1 -18134.153,E2 -18134.153} C_VEL
LIN {X 0,Y 264.06,Z 318.332,A -85,B 0,C 180,E1 -18138.289,E2 -18138.289} C_VEL
LIN {X 0,Y 263.621,Z 315.554,A -85,B 0,C 180,E1 -18142.181,E2 -18142.181} C_VEL
LIN {X 0,Y 263.255,Z 313.133,A -85,B 0,C 180,E1 -18145.901,E2 -18145.901} C_VEL
LIN {X 0,Y 263.127,Z 312.342,A -85,B 0,C 180,E1 -18147.711,E2 -18147.711} C_VEL
LIN {X 0,Y 263.19,Z 312.332,A -85,B 0,C 180,E1 -18151.785,E2 -18151.785} C_VEL
LIN {X 0,Y 263.22,Z 312.324,A -85,B 0,C 180,E1 -18155.2,E2 -18155.2} C_VEL
LIN {X 0,Y 263.258,Z 312.318,A -85,B 0,C 180,E1 -18159.693,E2 -18159.693} C_VEL
LIN {X 0,Y 263.339,Z 312.307,A -85,B 0,C 180,E1 -18164.521,E2 -18164.521} C_VEL
LIN {X 0,Y 263.343,Z 312.308,A -85,B 0,C 180,E1 -18169.233,E2 -18169.233} C_VEL
LIN {X 0,Y 263.52,Z 312.286,A -85,B 0,C 180,E1 -18172.337,E2 -18172.337} C_VEL
LIN {X 0,Y 263.743,Z 312.253,A -85,B 0,C 180,E1 -18178.473,E2 -18178.473} C_VEL
LIN {X 0,Y 263.743,Z 312.258,A -85,B 0,C 180,E1 -18181.527,E2 -18181.527} C_VEL
LIN {X 0,Y 263.52,Z 312.281,A -85,B 0,C 180,E1 -18187.663,E2 -18187.663} C_VEL
LIN {X 0,Y 263.343,Z 312.305,A -85,B 0,C 180,E1 -18190.767,E2 -18190.767} C_VEL
LIN {X 0,Y 263.339,Z 312.305,A -85,B 0,C 180,E1 -18195.479,E2 -18195.479} C_VEL
LIN {X 0,Y 263.258,Z 312.315,A -85,B 0,C 180,E1 -18200.307,E2 -18200.307} C_VEL
LIN {X 0,Y 263.203,Z 312.324,A -85,B 0,C 180,E1 -18205.292,E2 -18205.292} C_VEL
LIN {X 0,Y 263.161,Z 312.327,A -85,B 0,C 180,E1 -18208.732,E2 -18208.732} C_VEL
LIN {X 0,Y 263.128,Z 312.329,A -85,B 0,C 180,E1 -18212.289,E2 -18212.289} C_VEL
LIN {X 0,Y 263.198,Z 312.396,A -85,B 0,C 180,E1 -18216.77,E2 -18216.77} C_VEL
LIN {X 0,Y 263.441,Z 314.226,A -85,B 0,C 180,E1 -18219.812,E2 -18219.812} C_VEL
LIN {X 0,Y 263.811,Z 316.967,A -85,B 0,C 180,E1 -18224.006,E2 -18224.006} C_VEL
LIN {X 0,Y 263.931,Z 318.483,A -85,B 0,C 180,E1 -18226.187,E2 -18226.187} C_VEL
LIN {X 0,Y 263.93,Z 320.73,A -85,B 0,C 180,E1 -18229.036,E2 -18229.036} C_VEL
LIN {X 0,Y 264.92,Z 323.632,A -85,B 0,C 180,E1 -18229.337,E2 -18229.337} C_VEL
LIN {X 0,Y 266.326,Z 326.069,A -85,B 0,C 180,E1 -18229.698,E2 -18229.698} C_VEL
LIN {X 0,Y 272.078,Z 338.656,A -85,B 0,C 180,E1 -18231.365,E2 -18231.365} C_VEL
LIN {X 0,Y 276.79,Z 351.385,A -85,B 0,C 180,E1 -18233.031,E2 -18233.031} C_VEL
LIN {X 0,Y 280.539,Z 364.811,A -85,B 0,C 180,E1 -18234.818,E2 -18234.818} C_VEL
LIN {X 0,Y 283.193,Z 378.314,A -85,B 0,C 180,E1 -18236.698,E2 -18236.698} C_VEL
LIN {X 0,Y 284.115,Z 385.989,A -85,B 0,C 180,E1 -18237.81,E2 -18237.81} C_VEL
LIN {X 0,Y 281.133,Z 398.951,A -85,B 0,C 180,E1 -18239.381,E2 -18239.381} C_VEL
LIN {X 0,Y 278.244,Z 410.547,A -85,B 0,C 180,E1 -18241.115,E2 -18241.115} C_VEL
LIN {X 0,Y 275.254,Z 421.336,A -85,B 0,C 180,E1 -18243.055,E2 -18243.055} C_VEL
LIN {X 0,Y 272.427,Z 431.284,A -85,B 0,C 180,E1 -18245.216,E2 -18245.216} C_VEL
LIN {X 0,Y 269.435,Z 441.017,A -85,B 0,C 180,E1 -18247.777,E2 -18247.777} C_VEL
LIN {X 0,Y 266.955,Z 449.129,A -85,B 0,C 180,E1 -18250.388,E2 -18250.388} C_VEL
LIN {X 0,Y 265.011,Z 455.824,A -85,B 0,C 180,E1 -18253.04,E2 -18253.04} C_VEL
LIN {X 0,Y 263.314,Z 462.022,A -85,B 0,C 180,E1 -18256.102,E2 -18256.102} C_VEL
LIN {X 0,Y 262.147,Z 466.807,A -85,B 0,C 180,E1 -18259.184,E2 -18259.184} C_VEL
LIN {X 0,Y 261.406,Z 470.313,A -85,B 0,C 180,E1 -18262.275,E2 -18262.275} C_VEL
LIN {X 0,Y 261.097,Z 472.628,A -85,B 0,C 180,E1 -18265.369,E2 -18265.369} C_VEL
LIN {X 0,Y 261.049,Z 473.808,A -85,B 0,C 180,E1 -18268.458,E2 -18268.458} C_VEL
LIN {X 0,Y 261.05,Z 473.821,A -85,B 0,C 180,E1 -18271.543,E2 -18271.543} C_VEL
LIN {X 0,Y 261.1,Z 472.693,A -85,B 0,C 180,E1 -18274.632,E2 -18274.632} C_VEL
LIN {X 0,Y 261.405,Z 470.427,A -85,B 0,C 180,E1 -18277.726,E2 -18277.726} C_VEL
LIN {X 0,Y 262.106,Z 466.967,A -85,B 0,C 180,E1 -18280.819,E2 -18280.819} C_VEL
LIN {X 0,Y 263.294,Z 462.232,A -85,B 0,C 180,E1 -18283.901,E2 -18283.901} C_VEL
LIN {X 0,Y 264.928,Z 456.099,A -85,B 0,C 180,E1 -18286.967,E2 -18286.967} C_VEL
LIN {X 0,Y 267.197,Z 448.378,A -85,B 0,C 180,E1 -18289.995,E2 -18289.995} C_VEL
LIN {X 0,Y 269.7,Z 440.148,A -85,B 0,C 180,E1 -18292.605,E2 -18292.605} C_VEL
LIN {X 0,Y 272.802,Z 430.232,A -85,B 0,C 180,E1 -18295.156,E2 -18295.156} C_VEL
LIN {X 0,Y 275.659,Z 420.071,A -85,B 0,C 180,E1 -18297.317,E2 -18297.317} C_VEL
LIN {X 0,Y 278.976,Z 407.97,A -85,B 0,C 180,E1 -18299.423,E2 -18299.423} C_VEL
LIN {X 0,Y 281.991,Z 395.836,A -85,B 0,C 180,E1 -18301.141,E2 -18301.141} C_VEL
LIN {X 0,Y 284.119,Z 386.565,A -85,B 0,C 180,E1 -18302.238,E2 -18302.238} C_VEL
LIN {X 0,Y 283.359,Z 379.26,A -85,B 0,C 180,E1 -18303.292,E2 -18303.292} C_VEL
LIN {X 0,Y 281.299,Z 368.07,A -85,B 0,C 180,E1 -18304.866,E2 -18304.866} C_VEL
LIN {X 0,Y 278.339,Z 356.466,A -85,B 0,C 180,E1 -18306.423,E2 -18306.423} C_VEL
LIN {X 0,Y 273.969,Z 343.373,A -85,B 0,C 180,E1 -18308.148,E2 -18308.148} C_VEL
LIN {X 0,Y 269.339,Z 332.445,A -85,B 0,C 180,E1 -18309.594,E2 -18309.594} C_VEL
LIN {X 0,Y 265.545,Z 324.62,A -85,B 0,C 180,E1 -18310.645,E2 -18310.645} C_VEL
LIN {X 0,Y 264.105,Z 321.57,A -85,B 0,C 180,E1 -18311.042,E2 -18311.042} C_VEL
LIN {X 0,Y 263.914,Z 320.578,A -85,B 0,C 180,E1 -18311.139,E2 -18311.139} C_VEL
LIN {X 0,Y 263.954,Z 318.426,A -85,B 0,C 180,E1 -18314.036,E2 -18314.036} C_VEL
LIN {X 0,Y 263.797,Z 316.963,A -85,B 0,C 180,E1 -18316.157,E2 -18316.157} C_VEL
LIN {X 0,Y 263.412,Z 314.018,A -85,B 0,C 180,E1 -18320.691,E2 -18320.691} C_VEL
LIN {X 0,Y 263.202,Z 312.502,A -85,B 0,C 180,E1 -18323.231,E2 -18323.231} C_VEL
LIN {X 0,Y 263.128,Z 312.335,A -85,B 0,C 180,E1 -18327.711,E2 -18327.711} C_VEL
LIN {X 0,Y 263.148,Z 312.332,A -85,B 0,C 180,E1 -18331.805,E2 -18331.805} C_VEL
LIN {X 0,Y 263.189,Z 312.325,A -85,B 0,C 180,E1 -18335.218,E2 -18335.218} C_VEL
LIN {X 0,Y 263.262,Z 312.318,A -85,B 0,C 180,E1 -18339.693,E2 -18339.693} C_VEL
LIN {X 0,Y 263.35,Z 312.303,A -85,B 0,C 180,E1 -18344.522,E2 -18344.522} C_VEL
LIN {X 0,Y 263.349,Z 312.307,A -85,B 0,C 180,E1 -18349.233,E2 -18349.233} C_VEL
LIN {X 0,Y 263.525,Z 312.285,A -85,B 0,C 180,E1 -18352.337,E2 -18352.337} C_VEL
LIN {X 0,Y 263.748,Z 312.259,A -85,B 0,C 180,E1 -18358.473,E2 -18358.473} C_VEL
LIN {X 0,Y 263.748,Z 312.257,A -85,B 0,C 180,E1 -18361.527,E2 -18361.527} C_VEL
LIN {X 0,Y 263.525,Z 312.286,A -85,B 0,C 180,E1 -18367.663,E2 -18367.663} C_VEL
LIN {X 0,Y 263.352,Z 312.307,A -85,B 0,C 180,E1 -18370.766,E2 -18370.766} C_VEL
LIN {X 0,Y 263.32,Z 312.309,A -85,B 0,C 180,E1 -18375.087,E2 -18375.087} C_VEL
LIN {X 0,Y 262.7,Z 312.39,A -85,B 0,C 180,E1 -18376.363,E2 -18376.363} C_VEL
LIN {X 0,Y 259.811,Z 312.75,A -85,B 0,C 180,E1 -18378.44,E2 -18378.44} C_VEL
LIN {X 0,Y 257.302,Z 313.061,A -85,B 0,C 180,E1 -18380.13,E2 -18380.13} C_VEL
LIN {X 0,Y 256.197,Z 313.199,A -85,B 0,C 180,E1 -18381.443,E2 -18381.443} C_VEL
LIN {X 0,Y 256.095,Z 313.207,A -85,B 0,C 180,E1 -18381.888,E2 -18381.888} C_VEL
LIN {X 0,Y 256.128,Z 313.208,A -85,B 0,C 180,E1 -18386.042,E2 -18386.042} C_VEL
LIN {X 0,Y 256.103,Z 313.215,A -85,B 0,C 180,E1 -18389.601,E2 -18389.601} C_VEL
LIN {X 0,Y 256.082,Z 313.219,A -85,B 0,C 180,E1 -18391.704,E2 -18391.704} C_VEL
LIN {X 0,Y 256.39,Z 315.167,A -85,B 0,C 180,E1 -18395.144,E2 -18395.144} C_VEL
LIN {X 0,Y 256.78,Z 317.668,A -85,B 0,C 180,E1 -18399.013,E2 -18399.013} C_VEL
LIN {X 0,Y 257.19,Z 320.574,A -85,B 0,C 180,E1 -18403.09,E2 -18403.09} C_VEL
LIN {X 0,Y 257.404,Z 322.181,A -85,B 0,C 180,E1 -18405.225,E2 -18405.225} C_VEL
LIN {X 0,Y 257.369,Z 324.126,A -85,B 0,C 180,E1 -18407.628,E2 -18407.628} C_VEL
LIN {X 0,Y 258.556,Z 327.521,A -85,B 0,C 180,E1 -18408.018,E2 -18408.018} C_VEL
LIN {X 0,Y 259.859,Z 329.737,A -85,B 0,C 180,E1 -18408.371,E2 -18408.371} C_VEL
LIN {X 0,Y 265.229,Z 341.674,A -85,B 0,C 180,E1 -18410.01,E2 -18410.01} C_VEL
LIN {X 0,Y 270.182,Z 355.861,A -85,B 0,C 180,E1 -18411.9,E2 -18411.9} C_VEL
LIN {X 0,Y 273.658,Z 369.233,A -85,B 0,C 180,E1 -18413.714,E2 -18413.714} C_VEL
LIN {X 0,Y 275.764,Z 380.931,A -85,B 0,C 180,E1 -18415.355,E2 -18415.355} C_VEL
LIN {X 0,Y 277.076,Z 392.724,A -85,B 0,C 180,E1 -18417.103,E2 -18417.103} C_VEL
LIN {X 0,Y 276.83,Z 394.963,A -85,B 0,C 180,E1 -18417.409,E2 -18417.409} C_VEL
LIN {X 0,Y 273.591,Z 407.729,A -85,B 0,C 180,E1 -18419.085,E2 -18419.085} C_VEL
LIN {X 0,Y 270.556,Z 418.756,A -85,B 0,C 180,E1 -18420.853,E2 -18420.853} C_VEL
LIN {X 0,Y 267.29,Z 429.897,A -85,B 0,C 180,E1 -18423.027,E2 -18423.027} C_VEL
LIN {X 0,Y 264.493,Z 439.272,A -85,B 0,C 180,E1 -18425.26,E2 -18425.26} C_VEL
LIN {X 0,Y 261.501,Z 448.492,A -85,B 0,C 180,E1 -18427.898,E2 -18427.898} C_VEL
LIN {X 0,Y 258.792,Z 457.172,A -85,B 0,C 180,E1 -18430.981,E2 -18430.981} C_VEL
LIN {X 0,Y 256.789,Z 464.137,A -85,B 0,C 180,E1 -18434.116,E2 -18434.116} C_VEL
LIN {X 0,Y 255.32,Z 469.611,A -85,B 0,C 180,E1 -18437.278,E2 -18437.278} C_VEL
LIN {X 0,Y 254.486,Z 473.751,A -85,B 0,C 180,E1 -18440.462,E2 -18440.462} C_VEL
LIN {X 0,Y 254.046,Z 476.653,A -85,B 0,C 180,E1 -18443.646,E2 -18443.646} C_VEL
LIN {X 0,Y 253.9,Z 478.382,A -85,B 0,C 180,E1 -18446.826,E2 -18446.826} C_VEL
LIN {X 0,Y 253.979,Z 478.974,A -85,B 0,C 180,E1 -18449.999,E2 -18449.999} C_VEL
LIN {X 0,Y 253.901,Z 478.371,A -85,B 0,C 180,E1 -18453.173,E2 -18453.173} C_VEL
LIN {X 0,Y 254.045,Z 476.627,A -85,B 0,C 180,E1 -18456.352,E2 -18456.352} C_VEL
LIN {X 0,Y 254.485,Z 473.716,A -85,B 0,C 180,E1 -18459.537,E2 -18459.537} C_VEL
LIN {X 0,Y 255.318,Z 469.569,A -85,B 0,C 180,E1 -18462.721,E2 -18462.721} C_VEL
LIN {X 0,Y 256.798,Z 464.076,A -85,B 0,C 180,E1 -18465.882,E2 -18465.882} C_VEL
LIN {X 0,Y 258.789,Z 457.088,A -85,B 0,C 180,E1 -18469.018,E2 -18469.018} C_VEL
LIN {X 0,Y 261.475,Z 448.393,A -85,B 0,C 180,E1 -18472.103,E2 -18472.103} C_VEL
LIN {X 0,Y 264.515,Z 439.156,A -85,B 0,C 180,E1 -18474.737,E2 -18474.737} C_VEL
LIN {X 0,Y 267.332,Z 429.764,A -85,B 0,C 180,E1 -18476.967,E2 -18476.967} C_VEL
LIN {X 0,Y 270.58,Z 418.604,A -85,B 0,C 180,E1 -18479.143,E2 -18479.143} C_VEL
LIN {X 0,Y 273.941,Z 406.374,A -85,B 0,C 180,E1 -18481.084,E2 -18481.084} C_VEL
LIN {X 0,Y 277.079,Z 393.718,A -85,B 0,C 180,E1 -18482.71,E2 -18482.71} C_VEL
LIN {X 0,Y 275.638,Z 380.535,A -85,B 0,C 180,E1 -18484.672,E2 -18484.672} C_VEL
LIN {X 0,Y 273.182,Z 367.519,A -85,B 0,C 180,E1 -18486.491,E2 -18486.491} C_VEL
LIN {X 0,Y 269.725,Z 354.542,A -85,B 0,C 180,E1 -18488.236,E2 -18488.236} C_VEL
LIN {X 0,Y 264.96,Z 341.135,A -85,B 0,C 180,E1 -18490.027,E2 -18490.027} C_VEL
LIN {X 0,Y 260.766,Z 331.88,A -85,B 0,C 180,E1 -18491.31,E2 -18491.31} C_VEL
LIN {X 0,Y 259.12,Z 328.408,A -85,B 0,C 180,E1 -18491.779,E2 -18491.779} C_VEL
LIN {X 0,Y 257.606,Z 325.24,A -85,B 0,C 180,E1 -18492.217,E2 -18492.217} C_VEL
LIN {X 0,Y 257.353,Z 324.137,A -85,B 0,C 180,E1 -18492.325,E2 -18492.325} C_VEL
LIN {X 0,Y 257.358,Z 321.813,A -85,B 0,C 180,E1 -18495.234,E2 -18495.234} C_VEL
LIN {X 0,Y 256.979,Z 319.039,A -85,B 0,C 180,E1 -18498.977,E2 -18498.977} C_VEL
LIN {X 0,Y 256.575,Z 316.328,A -85,B 0,C 180,E1 -18502.943,E2 -18502.943} C_VEL
LIN {X 0,Y 256.172,Z 313.986,A -85,B 0,C 180,E1 -18506.723,E2 -18506.723} C_VEL
LIN {X 0,Y 256.087,Z 313.219,A -85,B 0,C 180,E1 -18508.572,E2 -18508.572} C_VEL
LIN {X 0,Y 256.133,Z 313.21,A -85,B 0,C 180,E1 -18512.195,E2 -18512.195} C_VEL
LIN {X 0,Y 256.161,Z 313.203,A -85,B 0,C 180,E1 -18515.699,E2 -18515.699} C_VEL
LIN {X 0,Y 256.161,Z 313.203,A -85,B 0,C 180,E1 -18519.105,E2 -18519.105} C_VEL
LIN {X 0,Y 256.289,Z 313.186,A -85,B 0,C 180,E1 -18524.085,E2 -18524.085} C_VEL
LIN {X 0,Y 256.285,Z 313.185,A -85,B 0,C 180,E1 -18528.933,E2 -18528.933} C_VEL
LIN {X 0,Y 256.462,Z 313.163,A -85,B 0,C 180,E1 -18532.125,E2 -18532.125} C_VEL
LIN {X 0,Y 256.49,Z 313.158,A -85,B 0,C 180,E1 -18536.859,E2 -18536.859} C_VEL
LIN {X 0,Y 256.744,Z 313.13,A -85,B 0,C 180,E1 -18540,E2 -18540} C_VEL
LIN {X 0,Y 256.49,Z 313.162,A -85,B 0,C 180,E1 -18543.142,E2 -18543.142} C_VEL
LIN {X 0,Y 256.462,Z 313.159,A -85,B 0,C 180,E1 -18547.876,E2 -18547.876} C_VEL
LIN {X 0,Y 256.285,Z 313.183,A -85,B 0,C 180,E1 -18551.067,E2 -18551.067} C_VEL
LIN {X 0,Y 256.289,Z 313.186,A -85,B 0,C 180,E1 -18555.916,E2 -18555.916} C_VEL
LIN {X 0,Y 256.162,Z 313.2,A -85,B 0,C 180,E1 -18560.896,E2 -18560.896} C_VEL
LIN {X 0,Y 256.183,Z 313.198,A -85,B 0,C 180,E1 -18565.139,E2 -18565.139} C_VEL
LIN {X 0,Y 256.099,Z 313.205,A -85,B 0,C 180,E1 -18569.602,E2 -18569.602} C_VEL
LIN {X 0,Y 256.063,Z 313.209,A -85,B 0,C 180,E1 -18573.294,E2 -18573.294} C_VEL
LIN {X 0,Y 256.078,Z 313.209,A -85,B 0,C 180,E1 -18575.194,E2 -18575.194} C_VEL
LIN {X 0,Y 256.238,Z 314.007,A -85,B 0,C 180,E1 -18577.309,E2 -18577.309} C_VEL
LIN {X 0,Y 256.523,Z 316.283,A -85,B 0,C 180,E1 -18581.112,E2 -18581.112} C_VEL
LIN {X 0,Y 256.873,Z 319.052,A -85,B 0,C 180,E1 -18585.345,E2 -18585.345} C_VEL
LIN {X 0,Y 256.894,Z 320.729,A -85,B 0,C 180,E1 -18587.654,E2 -18587.654} C_VEL
LIN {X 0,Y 258.02,Z 323.829,A -85,B 0,C 180,E1 -18588.011,E2 -18588.011} C_VEL
LIN {X 0,Y 259.454,Z 326.062,A -85,B 0,C 180,E1 -18588.393,E2 -18588.393} C_VEL
LIN {X 0,Y 265.469,Z 338.961,A -85,B 0,C 180,E1 -18590.23,E2 -18590.23} C_VEL
LIN {X 0,Y 270.034,Z 351.075,A -85,B 0,C 180,E1 -18591.912,E2 -18591.912} C_VEL
LIN {X 0,Y 274.037,Z 364.897,A -85,B 0,C 180,E1 -18593.854,E2 -18593.854} C_VEL
LIN {X 0,Y 276.48,Z 377.123,A -85,B 0,C 180,E1 -18595.62,E2 -18595.62} C_VEL
LIN {X 0,Y 277.835,Z 387.381,A -85,B 0,C 180,E1 -18597.171,E2 -18597.171} C_VEL
LIN {X 0,Y 274.716,Z 400.314,A -85,B 0,C 180,E1 -18598.8,E2 -18598.8} C_VEL
LIN {X 0,Y 271.427,Z 412.753,A -85,B 0,C 180,E1 -18600.744,E2 -18600.744} C_VEL
LIN {X 0,Y 268.41,Z 423.175,A -85,B 0,C 180,E1 -18602.73,E2 -18602.73} C_VEL
LIN {X 0,Y 265.479,Z 432.838,A -85,B 0,C 180,E1 -18604.941,E2 -18604.941} C_VEL
LIN {X 0,Y 262.425,Z 442.315,A -85,B 0,C 180,E1 -18607.566,E2 -18607.566} C_VEL
LIN {X 0,Y 259.571,Z 451.21,A -85,B 0,C 180,E1 -18610.631,E2 -18610.631} C_VEL
LIN {X 0,Y 257.653,Z 457.572,A -85,B 0,C 180,E1 -18613.358,E2 -18613.358} C_VEL
LIN {X 0,Y 255.982,Z 463.417,A -85,B 0,C 180,E1 -18616.505,E2 -18616.505} C_VEL
LIN {X 0,Y 255.12,Z 466.878,A -85,B 0,C 180,E1 -18618.883,E2 -18618.883} C_VEL
LIN {X 0,Y 254.35,Z 470.383,A -85,B 0,C 180,E1 -18622.06,E2 -18622.06} C_VEL
LIN {X 0,Y 254.014,Z 472.698,A -85,B 0,C 180,E1 -18625.239,E2 -18625.239} C_VEL
LIN {X 0,Y 253.96,Z 473.877,A -85,B 0,C 180,E1 -18628.415,E2 -18628.415} C_VEL
LIN {X 0,Y 253.96,Z 473.889,A -85,B 0,C 180,E1 -18631.586,E2 -18631.586} C_VEL
LIN {X 0,Y 254.086,Z 472.503,A -85,B 0,C 180,E1 -18635.278,E2 -18635.278} C_VEL
LIN {X 0,Y 254.349,Z 470.496,A -85,B 0,C 180,E1 -18637.942,E2 -18637.942} C_VEL
LIN {X 0,Y 255.085,Z 467.036,A -85,B 0,C 180,E1 -18641.12,E2 -18641.12} C_VEL
LIN {X 0,Y 256.362,Z 462.301,A -85,B 0,C 180,E1 -18644.284,E2 -18644.284} C_VEL
LIN {X 0,Y 258.099,Z 456.167,A -85,B 0,C 180,E1 -18647.43,E2 -18647.43} C_VEL
LIN {X 0,Y 260.51,Z 448.446,A -85,B 0,C 180,E1 -18650.531,E2 -18650.531} C_VEL
LIN {X 0,Y 263.122,Z 440.215,A -85,B 0,C 180,E1 -18653.202,E2 -18653.202} C_VEL
LIN {X 0,Y 266.284,Z 430.501,A -85,B 0,C 180,E1 -18655.761,E2 -18655.761} C_VEL
LIN {X 0,Y 269.352,Z 420.137,A -85,B 0,C 180,E1 -18658.012,E2 -18658.012} C_VEL
LIN {X 0,Y 272.75,Z 408.036,A -85,B 0,C 180,E1 -18660.163,E2 -18660.163} C_VEL
LIN {X 0,Y 275.909,Z 395.901,A -85,B 0,C 180,E1 -18661.907,E2 -18661.907} C_VEL
LIN {X 0,Y 277.859,Z 387.878,A -85,B 0,C 180,E1 -18662.883,E2 -18662.883} C_VEL
LIN {X 0,Y 276.463,Z 376.606,A -85,B 0,C 180,E1 -18664.578,E2 -18664.578} C_VEL
LIN {X 0,Y 273.968,Z 364.611,A -85,B 0,C 180,E1 -18666.317,E2 -18666.317} C_VEL
LIN {X 0,Y 270.175,Z 351.365,A -85,B 0,C 180,E1 -18668.175,E2 -18668.175} C_VEL
LIN {X 0,Y 265.97,Z 340.193,A -85,B 0,C 180,E1 -18669.734,E2 -18669.734} C_VEL
LIN {X 0,Y 260.793,Z 328.804,A -85,B 0,C 180,E1 -18671.37,E2 -18671.37} C_VEL
LIN {X 0,Y 258.744,Z 324.886,A -85,B 0,C 180,E1 -18671.942,E2 -18671.942} C_VEL
LIN {X 0,Y 257.159,Z 321.846,A -85,B 0,C 180,E1 -18672.394,E2 -18672.394} C_VEL
LIN {X 0,Y 256.888,Z 320.674,A -85,B 0,C 180,E1 -18672.495,E2 -18672.495} C_VEL
LIN {X 0,Y 256.848,Z 318.684,A -85,B 0,C 180,E1 -18675.351,E2 -18675.351} C_VEL
LIN {X 0,Y 256.534,Z 316.383,A -85,B 0,C 180,E1 -18678.89,E2 -18678.89} C_VEL
LIN {X 0,Y 256.235,Z 314,A -85,B 0,C 180,E1 -18682.885,E2 -18682.885} C_VEL
LIN {X 0,Y 256.105,Z 313.213,A -85,B 0,C 180,E1 -18685.412,E2 -18685.412} C_VEL
LIN {X 0,Y 256.082,Z 313.214,A -85,B 0,C 180,E1 -18688.571,E2 -18688.571} C_VEL
LIN {X 0,Y 256.093,Z 313.212,A -85,B 0,C 180,E1 -18692.19,E2 -18692.19} C_VEL
LIN {X 0,Y 256.133,Z 313.203,A -85,B 0,C 180,E1 -18695.695,E2 -18695.695} C_VEL
LIN {X 0,Y 256.162,Z 313.203,A -85,B 0,C 180,E1 -18699.104,E2 -18699.104} C_VEL
LIN {X 0,Y 256.299,Z 313.18,A -85,B 0,C 180,E1 -18704.085,E2 -18704.085} C_VEL
LIN {X 0,Y 256.29,Z 313.187,A -85,B 0,C 180,E1 -18708.933,E2 -18708.933} C_VEL
LIN {X 0,Y 256.467,Z 313.163,A -85,B 0,C 180,E1 -18712.125,E2 -18712.125} C_VEL
LIN {X 0,Y 256.494,Z 313.161,A -85,B 0,C 180,E1 -18716.858,E2 -18716.858} C_VEL
LIN {X 0,Y 256.742,Z 313.13,A -85,B 0,C 180,E1 -18720,E2 -18720} C_VEL
LIN {X 0,Y 256.494,Z 313.16,A -85,B 0,C 180,E1 -18723.141,E2 -18723.141} C_VEL
LIN {X 0,Y 256.489,Z 313.163,A -85,B 0,C 180,E1 -18727.874,E2 -18727.874} C_VEL
LIN {X 0,Y 256.294,Z 313.186,A -85,B 0,C 180,E1 -18731.066,E2 -18731.066} C_VEL
LIN {X 0,Y 256.299,Z 313.185,A -85,B 0,C 180,E1 -18735.915,E2 -18735.915} C_VEL
LIN {X 0,Y 256.161,Z 313.202,A -85,B 0,C 180,E1 -18740.895,E2 -18740.895} C_VEL
LIN {X 0,Y 256.095,Z 313.207,A -85,B 0,C 180,E1 -18741.888,E2 -18741.888} C_VEL
LIN {X 0,Y 255.405,Z 313.297,A -85,B 0,C 180,E1 -18743.201,E2 -18743.201} C_VEL
LIN {X 0,Y 252.587,Z 313.651,A -85,B 0,C 180,E1 -18745.343,E2 -18745.343} C_VEL
LIN {X 0,Y 250.204,Z 313.949,A -85,B 0,C 180,E1 -18747.085,E2 -18747.085} C_VEL
LIN {X 0,Y 249.168,Z 314.078,A -85,B 0,C 180,E1 -18748.435,E2 -18748.435} C_VEL
LIN {X 0,Y 249.075,Z 314.089,A -85,B 0,C 180,E1 -18748.893,E2 -18748.893} C_VEL
LIN {X 0,Y 249.047,Z 314.094,A -85,B 0,C 180,E1 -18750.527,E2 -18750.527} C_VEL
LIN {X 0,Y 249.335,Z 315.986,A -85,B 0,C 180,E1 -18754.315,E2 -18754.315} C_VEL
LIN {X 0,Y 249.693,Z 318.444,A -85,B 0,C 180,E1 -18758.259,E2 -18758.259} C_VEL
LIN {X 0,Y 250.129,Z 321.26,A -85,B 0,C 180,E1 -18762.403,E2 -18762.403} C_VEL
LIN {X 0,Y 250.398,Z 323.481,A -85,B 0,C 180,E1 -18765.438,E2 -18765.438} C_VEL
LIN {X 0,Y 250.395,Z 324.119,A -85,B 0,C 180,E1 -18766.17,E2 -18766.17} C_VEL
LIN {X 0,Y 251.319,Z 326.956,A -85,B 0,C 180,E1 -18766.493,E2 -18766.493} C_VEL
LIN {X 0,Y 253.053,Z 329.671,A -85,B 0,C 180,E1 -18766.986,E2 -18766.986} C_VEL
LIN {X 0,Y 258.773,Z 342.091,A -85,B 0,C 180,E1 -18768.834,E2 -18768.834} C_VEL
LIN {X 0,Y 263.177,Z 354.333,A -85,B 0,C 180,E1 -18770.576,E2 -18770.576} C_VEL
LIN {X 0,Y 266.546,Z 366.268,A -85,B 0,C 180,E1 -18772.28,E2 -18772.28} C_VEL
LIN {X 0,Y 269.055,Z 378.624,A -85,B 0,C 180,E1 -18774.072,E2 -18774.072} C_VEL
LIN {X 0,Y 270.549,Z 390.896,A -85,B 0,C 180,E1 -18775.951,E2 -18775.951} C_VEL
LIN {X 0,Y 270.807,Z 394.897,A -85,B 0,C 180,E1 -18776.59,E2 -18776.59} C_VEL
LIN {X 0,Y 267.502,Z 407.664,A -85,B 0,C 180,E1 -18778.301,E2 -18778.301} C_VEL
LIN {X 0,Y 264.325,Z 418.689,A -85,B 0,C 180,E1 -18780.097,E2 -18780.097} C_VEL
LIN {X 0,Y 260.936,Z 429.83,A -85,B 0,C 180,E1 -18782.315,E2 -18782.315} C_VEL
LIN {X 0,Y 258.006,Z 439.205,A -85,B 0,C 180,E1 -18784.594,E2 -18784.594} C_VEL
LIN {X 0,Y 254.858,Z 448.424,A -85,B 0,C 180,E1 -18787.29,E2 -18787.29} C_VEL
LIN {X 0,Y 252.353,Z 456.094,A -85,B 0,C 180,E1 -18790.052,E2 -18790.052} C_VEL
LIN {X 0,Y 250.379,Z 462.388,A -85,B 0,C 180,E1 -18792.825,E2 -18792.825} C_VEL
LIN {X 0,Y 248.75,Z 468.297,A -85,B 0,C 180,E1 -18796.104,E2 -18796.104} C_VEL
LIN {X 0,Y 247.842,Z 471.773,A -85,B 0,C 180,E1 -18798.55,E2 -18798.55} C_VEL
LIN {X 0,Y 247.154,Z 475.283,A -85,B 0,C 180,E1 -18801.826,E2 -18801.826} C_VEL
LIN {X 0,Y 246.838,Z 477.65,A -85,B 0,C 180,E1 -18805.219,E2 -18805.219} C_VEL
LIN {X 0,Y 246.852,Z 478.753,A -85,B 0,C 180,E1 -18808.368,E2 -18808.368} C_VEL
LIN {X 0,Y 246.889,Z 478.905,A -85,B 0,C 180,E1 -18809.999,E2 -18809.999} C_VEL
LIN {X 0,Y 246.806,Z 478.302,A -85,B 0,C 180,E1 -18813.264,E2 -18813.264} C_VEL
LIN {X 0,Y 246.966,Z 476.557,A -85,B 0,C 180,E1 -18816.535,E2 -18816.535} C_VEL
LIN {X 0,Y 247.432,Z 473.646,A -85,B 0,C 180,E1 -18819.812,E2 -18819.812} C_VEL
LIN {X 0,Y 248.357,Z 469.498,A -85,B 0,C 180,E1 -18823.083,E2 -18823.083} C_VEL
LIN {X 0,Y 249.922,Z 464.005,A -85,B 0,C 180,E1 -18826.331,E2 -18826.331} C_VEL
LIN {X 0,Y 252.031,Z 457.017,A -85,B 0,C 180,E1 -18829.549,E2 -18829.549} C_VEL
LIN {X 0,Y 254.844,Z 448.321,A -85,B 0,C 180,E1 -18832.71,E2 -18832.71} C_VEL
LIN {X 0,Y 258.026,Z 439.084,A -85,B 0,C 180,E1 -18835.402,E2 -18835.402} C_VEL
LIN {X 0,Y 260.971,Z 429.691,A -85,B 0,C 180,E1 -18837.68,E2 -18837.68} C_VEL
LIN {X 0,Y 264.635,Z 417.505,A -85,B 0,C 180,E1 -18840.083,E2 -18840.083} C_VEL
LIN {X 0,Y 268.193,Z 405.076,A -85,B 0,C 180,E1 -18842.048,E2 -18842.048} C_VEL
LIN {X 0,Y 270.732,Z 394.813,A -85,B 0,C 180,E1 -18843.394,E2 -18843.394} C_VEL
LIN {X 0,Y 269.465,Z 382.139,A -85,B 0,C 180,E1 -18845.367,E2 -18845.367} C_VEL
LIN {X 0,Y 267.207,Z 369.556,A -85,B 0,C 180,E1 -18847.223,E2 -18847.223} C_VEL
LIN {X 0,Y 264.201,Z 357.879,A -85,B 0,C 180,E1 -18848.887,E2 -18848.887} C_VEL
LIN {X 0,Y 259.878,Z 345.016,A -85,B 0,C 180,E1 -18850.699,E2 -18850.699} C_VEL
LIN {X 0,Y 254.41,Z 332.598,A -85,B 0,C 180,E1 -18852.543,E2 -18852.543} C_VEL
LIN {X 0,Y 252.52,Z 328.735,A -85,B 0,C 180,E1 -18853.111,E2 -18853.111} C_VEL
LIN {X 0,Y 250.772,Z 325.712,A -85,B 0,C 180,E1 -18853.624,E2 -18853.624} C_VEL
LIN {X 0,Y 250.364,Z 324.032,A -85,B 0,C 180,E1 -18853.823,E2 -18853.823} C_VEL
LIN {X 0,Y 250.198,Z 321.711,A -85,B 0,C 180,E1 -18856.912,E2 -18856.912} C_VEL
LIN {X 0,Y 249.894,Z 319.754,A -85,B 0,C 180,E1 -18859.696,E2 -18859.696} C_VEL
LIN {X 0,Y 249.481,Z 317.133,A -85,B 0,C 180,E1 -18863.731,E2 -18863.731} C_VEL
LIN {X 0,Y 249.113,Z 314.719,A -85,B 0,C 180,E1 -18867.816,E2 -18867.816} C_VEL
LIN {X 0,Y 249.042,Z 314.097,A -85,B 0,C 180,E1 -18869.472,E2 -18869.472} C_VEL
LIN {X 0,Y 249.067,Z 314.088,A -85,B 0,C 180,E1 -18873.162,E2 -18873.162} C_VEL
LIN {X 0,Y 249.074,Z 314.084,A -85,B 0,C 180,E1 -18876.732,E2 -18876.732} C_VEL
LIN {X 0,Y 249.105,Z 314.079,A -85,B 0,C 180,E1 -18880.211,E2 -18880.211} C_VEL
LIN {X 0,Y 249.237,Z 314.065,A -85,B 0,C 180,E1 -18883.622,E2 -18883.622} C_VEL
LIN {X 0,Y 249.232,Z 314.062,A -85,B 0,C 180,E1 -18888.616,E2 -18888.616} C_VEL
LIN {X 0,Y 249.411,Z 314.041,A -85,B 0,C 180,E1 -18891.901,E2 -18891.901} C_VEL
LIN {X 0,Y 249.281,Z 314.056,A -85,B 0,C 180,E1 -18895.148,E2 -18895.148} C_VEL
LIN {X 0,Y 249.668,Z 314.006,A -85,B 0,C 180,E1 -18898.387,E2 -18898.387} C_VEL
LIN {X 0,Y 249.668,Z 314.011,A -85,B 0,C 180,E1 -18901.613,E2 -18901.613} C_VEL
LIN {X 0,Y 249.42,Z 314.042,A -85,B 0,C 180,E1 -18906.531,E2 -18906.531} C_VEL
LIN {X 0,Y 249.337,Z 314.053,A -85,B 0,C 180,E1 -18909.737,E2 -18909.737} C_VEL
LIN {X 0,Y 249.195,Z 314.065,A -85,B 0,C 180,E1 -18914.704,E2 -18914.704} C_VEL
LIN {X 0,Y 249.134,Z 314.073,A -85,B 0,C 180,E1 -18918.078,E2 -18918.078} C_VEL
LIN {X 0,Y 249.082,Z 314.085,A -85,B 0,C 180,E1 -18921.519,E2 -18921.519} C_VEL
LIN {X 0,Y 249.126,Z 314.077,A -85,B 0,C 180,E1 -18925.483,E2 -18925.483} C_VEL
LIN {X 0,Y 249.068,Z 314.081,A -85,B 0,C 180,E1 -18928.99,E2 -18928.99} C_VEL
LIN {X 0,Y 249.026,Z 314.086,A -85,B 0,C 180,E1 -18932.427,E2 -18932.427} C_VEL
LIN {X 0,Y 249.041,Z 314.101,A -85,B 0,C 180,E1 -18935.079,E2 -18935.079} C_VEL
LIN {X 0,Y 249.32,Z 315.876,A -85,B 0,C 180,E1 -18938.327,E2 -18938.327} C_VEL
LIN {X 0,Y 249.661,Z 318.369,A -85,B 0,C 180,E1 -18942.501,E2 -18942.501} C_VEL
LIN {X 0,Y 249.86,Z 320.743,A -85,B 0,C 180,E1 -18946.133,E2 -18946.133} C_VEL
LIN {X 0,Y 251.102,Z 324.063,A -85,B 0,C 180,E1 -18946.58,E2 -18946.58} C_VEL
LIN {X 0,Y 252.645,Z 326.353,A -85,B 0,C 180,E1 -18947.015,E2 -18947.015} C_VEL
LIN {X 0,Y 257.064,Z 335.202,A -85,B 0,C 180,E1 -18948.4,E2 -18948.4} C_VEL
LIN {X 0,Y 261.854,Z 346.665,A -85,B 0,C 180,E1 -18950.124,E2 -18950.124} C_VEL
LIN {X 0,Y 266.219,Z 359.949,A -85,B 0,C 180,E1 -18952.079,E2 -18952.079} C_VEL
LIN {X 0,Y 269.281,Z 372.802,A -85,B 0,C 180,E1 -18954.006,E2 -18954.006} C_VEL
LIN {X 0,Y 271.232,Z 385.677,A -85,B 0,C 180,E1 -18956.013,E2 -18956.013} C_VEL
LIN {X 0,Y 271.538,Z 388.671,A -85,B 0,C 180,E1 -18956.492,E2 -18956.492} C_VEL
LIN {X 0,Y 268.324,Z 401.634,A -85,B 0,C 180,E1 -18958.19,E2 -18958.19} C_VEL
LIN {X 0,Y 264.922,Z 413.867,A -85,B 0,C 180,E1 -18960.172,E2 -18960.172} C_VEL
LIN {X 0,Y 261.703,Z 424.534,A -85,B 0,C 180,E1 -18962.285,E2 -18962.285} C_VEL
LIN {X 0,Y 258.556,Z 434.391,A -85,B 0,C 180,E1 -18964.653,E2 -18964.653} C_VEL
LIN {X 0,Y 255.839,Z 442.387,A -85,B 0,C 180,E1 -18966.956,E2 -18966.956} C_VEL
LIN {X 0,Y 253.171,Z 450.277,A -85,B 0,C 180,E1 -18969.697,E2 -18969.697} C_VEL
LIN {X 0,Y 250.82,Z 457.643,A -85,B 0,C 180,E1 -18972.891,E2 -18972.891} C_VEL
LIN {X 0,Y 249.046,Z 463.487,A -85,B 0,C 180,E1 -18976.122,E2 -18976.122} C_VEL
LIN {X 0,Y 248.115,Z 466.948,A -85,B 0,C 180,E1 -18978.564,E2 -18978.564} C_VEL
LIN {X 0,Y 247.294,Z 470.452,A -85,B 0,C 180,E1 -18981.831,E2 -18981.831} C_VEL
LIN {X 0,Y 246.923,Z 472.767,A -85,B 0,C 180,E1 -18985.102,E2 -18985.102} C_VEL
LIN {X 0,Y 246.873,Z 473.946,A -85,B 0,C 180,E1 -18988.369,E2 -18988.369} C_VEL
LIN {X 0,Y 246.873,Z 473.958,A -85,B 0,C 180,E1 -18991.632,E2 -18991.632} C_VEL
LIN {X 0,Y 246.983,Z 472.701,A -85,B 0,C 180,E1 -18995.164,E2 -18995.164} C_VEL
LIN {X 0,Y 247.292,Z 470.564,A -85,B 0,C 180,E1 -18998.17,E2 -18998.17} C_VEL
LIN {X 0,Y 248.086,Z 467.104,A -85,B 0,C 180,E1 -19001.438,E2 -19001.438} C_VEL
LIN {X 0,Y 249.432,Z 462.369,A -85,B 0,C 180,E1 -19004.69,E2 -19004.69} C_VEL
LIN {X 0,Y 251.401,Z 455.816,A -85,B 0,C 180,E1 -19008.105,E2 -19008.105} C_VEL
LIN {X 0,Y 253.816,Z 448.513,A -85,B 0,C 180,E1 -19011.098,E2 -19011.098} C_VEL
LIN {X 0,Y 256.548,Z 440.282,A -85,B 0,C 180,E1 -19013.833,E2 -19013.833} C_VEL
LIN {X 0,Y 259.769,Z 430.853,A -85,B 0,C 180,E1 -19016.375,E2 -19016.375} C_VEL
LIN {X 0,Y 263.059,Z 420.203,A -85,B 0,C 180,E1 -19018.744,E2 -19018.744} C_VEL
LIN {X 0,Y 266.607,Z 408.101,A -85,B 0,C 180,E1 -19020.933,E2 -19020.933} C_VEL
LIN {X 0,Y 269.911,Z 395.966,A -85,B 0,C 180,E1 -19022.704,E2 -19022.704} C_VEL
LIN {X 0,Y 271.573,Z 389.158,A -85,B 0,C 180,E1 -19023.557,E2 -19023.557} C_VEL
LIN {X 0,Y 270.091,Z 377.205,A -85,B 0,C 180,E1 -19025.446,E2 -19025.446} C_VEL
LIN {X 0,Y 267.475,Z 364.543,A -85,B 0,C 180,E1 -19027.36,E2 -19027.36} C_VEL
LIN {X 0,Y 264.109,Z 352.987,A -85,B 0,C 180,E1 -19029.079,E2 -19029.079} C_VEL
LIN {X 0,Y 259.863,Z 341.49,A -85,B 0,C 180,E1 -19030.776,E2 -19030.776} C_VEL
LIN {X 0,Y 254.53,Z 329.856,A -85,B 0,C 180,E1 -19032.571,E2 -19032.571} C_VEL
LIN {X 0,Y 252.519,Z 326.023,A -85,B 0,C 180,E1 -19033.175,E2 -19033.175} C_VEL
LIN {X 0,Y 250.344,Z 322.491,A -85,B 0,C 180,E1 -19033.808,E2 -19033.808} C_VEL
LIN {X 0,Y 249.878,Z 320.729,A -85,B 0,C 180,E1 -19034.038,E2 -19034.038} C_VEL
LIN {X 0,Y 249.671,Z 318.467,A -85,B 0,C 180,E1 -19037.501,E2 -19037.501} C_VEL
LIN {X 0,Y 249.332,Z 315.978,A -85,B 0,C 180,E1 -19041.675,E2 -19041.675} C_VEL
LIN {X 0,Y 249.081,Z 314.208,A -85,B 0,C 180,E1 -19044.91,E2 -19044.91} C_VEL
LIN {X 0,Y 249.002,Z 314.093,A -85,B 0,C 180,E1 -19049.466,E2 -19049.466} C_VEL
LIN {X 0,Y 249.035,Z 314.087,A -85,B 0,C 180,E1 -19053.158,E2 -19053.158} C_VEL
LIN {X 0,Y 249.055,Z 314.088,A -85,B 0,C 180,E1 -19056.73,E2 -19056.73} C_VEL
LIN {X 0,Y 249.108,Z 314.077,A -85,B 0,C 180,E1 -19060.211,E2 -19060.211} C_VEL
LIN {X 0,Y 249.242,Z 314.058,A -85,B 0,C 180,E1 -19063.622,E2 -19063.622} C_VEL
LIN {X 0,Y 249.234,Z 314.065,A -85,B 0,C 180,E1 -19068.616,E2 -19068.616} C_VEL
LIN {X 0,Y 249.417,Z 314.041,A -85,B 0,C 180,E1 -19071.901,E2 -19071.901} C_VEL
LIN {X 0,Y 249.284,Z 314.059,A -85,B 0,C 180,E1 -19075.148,E2 -19075.148} C_VEL
LIN {X 0,Y 249.673,Z 314.011,A -85,B 0,C 180,E1 -19078.387,E2 -19078.387} C_VEL
LIN {X 0,Y 249.673,Z 314.01,A -85,B 0,C 180,E1 -19081.613,E2 -19081.613} C_VEL
LIN {X 0,Y 249.431,Z 314.04,A -85,B 0,C 180,E1 -19086.471,E2 -19086.471} C_VEL
LIN {X 0,Y 249.342,Z 314.052,A -85,B 0,C 180,E1 -19089.736,E2 -19089.736} C_VEL
LIN {X 0,Y 249.204,Z 314.069,A -85,B 0,C 180,E1 -19094.703,E2 -19094.703} C_VEL
LIN {X 0,Y 249.137,Z 314.077,A -85,B 0,C 180,E1 -19098.077,E2 -19098.077} C_VEL
LIN {X 0,Y 249.06,Z 314.086,A -85,B 0,C 180,E1 -19101.869,E2 -19101.869} C_VEL
LIN {X 0,Y 249.116,Z 314.079,A -85,B 0,C 180,E1 -19105.475,E2 -19105.475} C_VEL
LIN {X 0,Y 249.075,Z 314.089,A -85,B 0,C 180,E1 -19108.893,E2 -19108.893} C_VEL
LIN {X 0,Y 248.42,Z 314.361,A -85,B 0,C 180,E1 -19110.241,E2 -19110.241} C_VEL
LIN {X 0,Y 245.734,Z 315.649,A -85,B 0,C 180,E1 -19112.432,E2 -19112.432} C_VEL
LIN {X 0,Y 243.488,Z 317.044,A -85,B 0,C 180,E1 -19114.208,E2 -19114.208} C_VEL
LIN {X 0,Y 242.558,Z 318.044,A -85,B 0,C 180,E1 -19115.582,E2 -19115.582} C_VEL
LIN {X 0,Y 242.498,Z 318.342,A -85,B 0,C 180,E1 -19116.048,E2 -19116.048} C_VEL
LIN {X 0,Y 242.818,Z 320.543,A -85,B 0,C 180,E1 -19119.55,E2 -19119.55} C_VEL
LIN {X 0,Y 243.264,Z 323.497,A -85,B 0,C 180,E1 -19123.897,E2 -19123.897} C_VEL
LIN {X 0,Y 243.351,Z 323.945,A -85,B 0,C 180,E1 -19124.527,E2 -19124.527} C_VEL
LIN {X 0,Y 244.396,Z 327,A -85,B 0,C 180,E1 -19124.937,E2 -19124.937} C_VEL
LIN {X 0,Y 246.174,Z 329.723,A -85,B 0,C 180,E1 -19125.479,E2 -19125.479} C_VEL
LIN {X 0,Y 248.261,Z 333.591,A -85,B 0,C 180,E1 -19126.142,E2 -19126.142} C_VEL
LIN {X 0,Y 253.722,Z 345.885,A -85,B 0,C 180,E1 -19128.11,E2 -19128.11} C_VEL
LIN {X 0,Y 257.904,Z 358.231,A -85,B 0,C 180,E1 -19129.969,E2 -19129.969} C_VEL
LIN {X 0,Y 260.988,Z 369.895,A -85,B 0,C 180,E1 -19131.731,E2 -19131.731} C_VEL
LIN {X 0,Y 263.351,Z 383.505,A -85,B 0,C 180,E1 -19133.83,E2 -19133.83} C_VEL
LIN {X 0,Y 264.402,Z 394.447,A -85,B 0,C 180,E1 -19135.609,E2 -19135.609} C_VEL
LIN {X 0,Y 264.311,Z 397.306,A -85,B 0,C 180,E1 -19136.055,E2 -19136.055} C_VEL
LIN {X 0,Y 260.783,Z 409.947,A -85,B 0,C 180,E1 -19137.842,E2 -19137.842} C_VEL
LIN {X 0,Y 257.563,Z 420.577,A -85,B 0,C 180,E1 -19139.682,E2 -19139.682} C_VEL
LIN {X 0,Y 254.043,Z 431.393,A -85,B 0,C 180,E1 -19141.946,E2 -19141.946} C_VEL
LIN {X 0,Y 251.079,Z 440.57,A -85,B 0,C 180,E1 -19144.287,E2 -19144.287} C_VEL
LIN {X 0,Y 247.865,Z 449.569,A -85,B 0,C 180,E1 -19147.053,E2 -19147.053} C_VEL
LIN {X 0,Y 245.288,Z 457.036,A -85,B 0,C 180,E1 -19149.89,E2 -19149.89} C_VEL
LIN {X 0,Y 243.054,Z 464,A -85,B 0,C 180,E1 -19153.192,E2 -19153.192} C_VEL
LIN {X 0,Y 241.415,Z 469.474,A -85,B 0,C 180,E1 -19156.532,E2 -19156.532} C_VEL
LIN {X 0,Y 240.399,Z 473.614,A -85,B 0,C 180,E1 -19159.897,E2 -19159.897} C_VEL
LIN {X 0,Y 239.889,Z 476.515,A -85,B 0,C 180,E1 -19163.27,E2 -19163.27} C_VEL
LIN {X 0,Y 239.714,Z 478.245,A -85,B 0,C 180,E1 -19166.638,E2 -19166.638} C_VEL
LIN {X 0,Y 239.801,Z 478.836,A -85,B 0,C 180,E1 -19169.999,E2 -19169.999} C_VEL
LIN {X 0,Y 239.714,Z 478.233,A -85,B 0,C 180,E1 -19173.361,E2 -19173.361} C_VEL
LIN {X 0,Y 239.888,Z 476.488,A -85,B 0,C 180,E1 -19176.729,E2 -19176.729} C_VEL
LIN {X 0,Y 240.398,Z 473.575,A -85,B 0,C 180,E1 -19180.102,E2 -19180.102} C_VEL
LIN {X 0,Y 241.413,Z 469.428,A -85,B 0,C 180,E1 -19183.467,E2 -19183.467} C_VEL
LIN {X 0,Y 243.063,Z 463.935,A -85,B 0,C 180,E1 -19186.806,E2 -19186.806} C_VEL
LIN {X 0,Y 245.283,Z 456.945,A -85,B 0,C 180,E1 -19190.109,E2 -19190.109} C_VEL
LIN {X 0,Y 248.248,Z 448.249,A -85,B 0,C 180,E1 -19193.349,E2 -19193.349} C_VEL
LIN {X 0,Y 251.568,Z 439.012,A -85,B 0,C 180,E1 -19196.103,E2 -19196.103} C_VEL
LIN {X 0,Y 254.658,Z 429.619,A -85,B 0,C 180,E1 -19198.427,E2 -19198.427} C_VEL
LIN {X 0,Y 258.155,Z 418.458,A -85,B 0,C 180,E1 -19200.692,E2 -19200.692} C_VEL
LIN {X 0,Y 261.832,Z 406.228,A -85,B 0,C 180,E1 -19202.695,E2 -19202.695} C_VEL
LIN {X 0,Y 264.308,Z 397.059,A -85,B 0,C 180,E1 -19203.944,E2 -19203.944} C_VEL
LIN {X 0,Y 263.795,Z 388.045,A -85,B 0,C 180,E1 -19205.411,E2 -19205.411} C_VEL
LIN {X 0,Y 262,Z 375.539,A -85,B 0,C 180,E1 -19207.377,E2 -19207.377} C_VEL
LIN {X 0,Y 259.141,Z 362.729,A -85,B 0,C 180,E1 -19209.32,E2 -19209.32} C_VEL
LIN {X 0,Y 254.968,Z 349.274,A -85,B 0,C 180,E1 -19211.332,E2 -19211.332} C_VEL
LIN {X 0,Y 249.88,Z 337.144,A -85,B 0,C 180,E1 -19213.229,E2 -19213.229} C_VEL
LIN {X 0,Y 247.633,Z 332.713,A -85,B 0,C 180,E1 -19213.988,E2 -19213.988} C_VEL
LIN {X 0,Y 245.579,Z 328.676,A -85,B 0,C 180,E1 -19214.644,E2 -19214.644} C_VEL
LIN {X 0,Y 243.902,Z 325.936,A -85,B 0,C 180,E1 -19215.166,E2 -19215.166} C_VEL
LIN {X 0,Y 243.348,Z 323.957,A -85,B 0,C 180,E1 -19215.4,E2 -19215.4} C_VEL
LIN {X 0,Y 242.998,Z 321.606,A -85,B 0,C 180,E1 -19218.76,E2 -19218.76} C_VEL
LIN {X 0,Y 242.624,Z 319.164,A -85,B 0,C 180,E1 -19222.534,E2 -19222.534} C_VEL
LIN {X 0,Y 242.241,Z 316.79,A -85,B 0,C 180,E1 -19226.548,E2 -19226.548} C_VEL
LIN {X 0,Y 242.002,Z 314.973,A -85,B 0,C 180,E1 -19230.416,E2 -19230.416} C_VEL
LIN {X 0,Y 242.063,Z 314.96,A -85,B 0,C 180,E1 -19234.183,E2 -19234.183} C_VEL
LIN {X 0,Y 242.048,Z 314.958,A -85,B 0,C 180,E1 -19238.297,E2 -19238.297} C_VEL
LIN {X 0,Y 242.158,Z 314.944,A -85,B 0,C 180,E1 -19243.278,E2 -19243.278} C_VEL
LIN {X 0,Y 242.169,Z 314.941,A -85,B 0,C 180,E1 -19248.279,E2 -19248.279} C_VEL
LIN {X 0,Y 242.365,Z 314.917,A -85,B 0,C 180,E1 -19251.664,E2 -19251.664} C_VEL
LIN {X 0,Y 242.24,Z 314.932,A -85,B 0,C 180,E1 -19255.007,E2 -19255.007} C_VEL
LIN {X 0,Y 242.629,Z 314.882,A -85,B 0,C 180,E1 -19258.34,E2 -19258.34} C_VEL
LIN {X 0,Y 242.629,Z 314.888,A -85,B 0,C 180,E1 -19261.66,E2 -19261.66} C_VEL
LIN {X 0,Y 242.394,Z 314.917,A -85,B 0,C 180,E1 -19266.66,E2 -19266.66} C_VEL
LIN {X 0,Y 242.261,Z 314.934,A -85,B 0,C 180,E1 -19270.024,E2 -19270.024} C_VEL
LIN {X 0,Y 242.158,Z 314.942,A -85,B 0,C 180,E1 -19275.142,E2 -19275.142} C_VEL
LIN {X 0,Y 242.068,Z 314.957,A -85,B 0,C 180,E1 -19278.625,E2 -19278.625} C_VEL
LIN {X 0,Y 242.008,Z 314.965,A -85,B 0,C 180,E1 -19282.181,E2 -19282.181} C_VEL
LIN {X 0,Y 242.062,Z 314.956,A -85,B 0,C 180,E1 -19285.839,E2 -19285.839} C_VEL
LIN {X 0,Y 242.003,Z 314.961,A -85,B 0,C 180,E1 -19289.584,E2 -19289.584} C_VEL
LIN {X 0,Y 241.976,Z 314.964,A -85,B 0,C 180,E1 -19293.493,E2 -19293.493} C_VEL
LIN {X 0,Y 242.106,Z 315.718,A -85,B 0,C 180,E1 -19295.632,E2 -19295.632} C_VEL
LIN {X 0,Y 242.411,Z 317.891,A -85,B 0,C 180,E1 -19299.63,E2 -19299.63} C_VEL
LIN {X 0,Y 242.779,Z 320.695,A -85,B 0,C 180,E1 -19304.297,E2 -19304.297} C_VEL
LIN {X 0,Y 242.874,Z 321.048,A -85,B 0,C 180,E1 -19304.565,E2 -19304.565} C_VEL
LIN {X 0,Y 244.08,Z 324.137,A -85,B 0,C 180,E1 -19304.996,E2 -19304.996} C_VEL
LIN {X 0,Y 245.792,Z 326.567,A -85,B 0,C 180,E1 -19305.512,E2 -19305.512} C_VEL
LIN {X 0,Y 247.867,Z 330.354,A -85,B 0,C 180,E1 -19306.175,E2 -19306.175} C_VEL
LIN {X 0,Y 252.419,Z 339.855,A -85,B 0,C 180,E1 -19307.769,E2 -19307.769} C_VEL
LIN {X 0,Y 256.981,Z 351.322,A -85,B 0,C 180,E1 -19309.599,E2 -19309.599} C_VEL
LIN {X 0,Y 260.587,Z 363.194,A -85,B 0,C 180,E1 -19311.456,E2 -19311.456} C_VEL
LIN {X 0,Y 263.433,Z 376.03,A -85,B 0,C 180,E1 -19313.484,E2 -19313.484} C_VEL
LIN {X 0,Y 265.144,Z 388.752,A -85,B 0,C 180,E1 -19315.572,E2 -19315.572} C_VEL
LIN {X 0,Y 265.141,Z 391.192,A -85,B 0,C 180,E1 -19315.966,E2 -19315.966} C_VEL
LIN {X 0,Y 261.636,Z 404.049,A -85,B 0,C 180,E1 -19317.733,E2 -19317.733} C_VEL
LIN {X 0,Y 258.131,Z 415.888,A -85,B 0,C 180,E1 -19319.757,E2 -19319.757} C_VEL
LIN {X 0,Y 254.704,Z 426.723,A -85,B 0,C 180,E1 -19322.027,E2 -19322.027} C_VEL
LIN {X 0,Y 251.624,Z 435.914,A -85,B 0,C 180,E1 -19324.348,E2 -19324.348} C_VEL
LIN {X 0,Y 248.418,Z 444.906,A -85,B 0,C 180,E1 -19327.109,E2 -19327.109} C_VEL
LIN {X 0,Y 245.772,Z 452.358,A -85,B 0,C 180,E1 -19329.932,E2 -19329.932} C_VEL
LIN {X 0,Y 243.454,Z 459.322,A -85,B 0,C 180,E1 -19333.222,E2 -19333.222} C_VEL
LIN {X 0,Y 241.697,Z 464.795,A -85,B 0,C 180,E1 -19336.549,E2 -19336.549} C_VEL
LIN {X 0,Y 240.639,Z 468.924,A -85,B 0,C 180,E1 -19339.909,E2 -19339.909} C_VEL
LIN {X 0,Y 240.02,Z 471.824,A -85,B 0,C 180,E1 -19343.275,E2 -19343.275} C_VEL
LIN {X 0,Y 239.78,Z 473.566,A -85,B 0,C 180,E1 -19346.64,E2 -19346.64} C_VEL
LIN {X 0,Y 239.805,Z 474.172,A -85,B 0,C 180,E1 -19350.001,E2 -19350.001} C_VEL
LIN {X 0,Y 239.781,Z 473.603,A -85,B 0,C 180,E1 -19353.361,E2 -19353.361} C_VEL
LIN {X 0,Y 239.997,Z 471.911,A -85,B 0,C 180,E1 -19356.727,E2 -19356.727} C_VEL
LIN {X 0,Y 240.627,Z 469.056,A -85,B 0,C 180,E1 -19360.093,E2 -19360.093} C_VEL
LIN {X 0,Y 241.676,Z 464.972,A -85,B 0,C 180,E1 -19363.453,E2 -19363.453} C_VEL
LIN {X 0,Y 243.394,Z 459.556,A -85,B 0,C 180,E1 -19366.784,E2 -19366.784} C_VEL
LIN {X 0,Y 245.699,Z 452.656,A -85,B 0,C 180,E1 -19370.075,E2 -19370.075} C_VEL
LIN {X 0,Y 248.76,Z 444.044,A -85,B 0,C 180,E1 -19373.299,E2 -19373.299} C_VEL
LIN {X 0,Y 251.56,Z 436.303,A -85,B 0,C 180,E1 -19375.66,E2 -19375.66} C_VEL
LIN {X 0,Y 255.112,Z 425.567,A -85,B 0,C 180,E1 -19378.374,E2 -19378.374} C_VEL
LIN {X 0,Y 258.977,Z 413.501,A -85,B 0,C 180,E1 -19380.812,E2 -19380.812} C_VEL
LIN {X 0,Y 262.54,Z 401.179,A -85,B 0,C 180,E1 -19382.825,E2 -19382.825} C_VEL
LIN {X 0,Y 265.306,Z 390.428,A -85,B 0,C 180,E1 -19384.265,E2 -19384.265} C_VEL
LIN {X 0,Y 263.803,Z 378.2,A -85,B 0,C 180,E1 -19386.299,E2 -19386.299} C_VEL
LIN {X 0,Y 261.438,Z 366.32,A -85,B 0,C 180,E1 -19388.191,E2 -19388.191} C_VEL
LIN {X 0,Y 257.701,Z 353.361,A -85,B 0,C 180,E1 -19390.216,E2 -19390.216} C_VEL
LIN {X 0,Y 253.257,Z 341.677,A -85,B 0,C 180,E1 -19392.07,E2 -19392.07} C_VEL
LIN {X 0,Y 249.47,Z 333.592,A -85,B 0,C 180,E1 -19393.423,E2 -19393.423} C_VEL
LIN {X 0,Y 247.306,Z 329.509,A -85,B 0,C 180,E1 -19394.153,E2 -19394.153} C_VEL
LIN {X 0,Y 245.285,Z 325.642,A -85,B 0,C 180,E1 -19394.803,E2 -19394.803} C_VEL
LIN {X 0,Y 243.481,Z 322.979,A -85,B 0,C 180,E1 -19395.358,E2 -19395.358} C_VEL
LIN {X 0,Y 242.827,Z 320.828,A -85,B 0,C 180,E1 -19395.642,E2 -19395.642} C_VEL
LIN {X 0,Y 242.417,Z 317.994,A -85,B 0,C 180,E1 -19400.371,E2 -19400.371} C_VEL
LIN {X 0,Y 242.133,Z 315.741,A -85,B 0,C 180,E1 -19404.514,E2 -19404.514} C_VEL
LIN {X 0,Y 241.979,Z 314.971,A -85,B 0,C 180,E1 -19406.507,E2 -19406.507} C_VEL
LIN {X 0,Y 241.977,Z 314.969,A -85,B 0,C 180,E1 -19410.612,E2 -19410.612} C_VEL
LIN {X 0,Y 242.032,Z 314.963,A -85,B 0,C 180,E1 -19414.179,E2 -19414.179} C_VEL
LIN {X 0,Y 242.025,Z 314.959,A -85,B 0,C 180,E1 -19418.314,E2 -19418.314} C_VEL
LIN {X 0,Y 242.163,Z 314.941,A -85,B 0,C 180,E1 -19423.278,E2 -19423.278} C_VEL
LIN {X 0,Y 242.149,Z 314.941,A -85,B 0,C 180,E1 -19426.574,E2 -19426.574} C_VEL
LIN {X 0,Y 242.341,Z 314.923,A -85,B 0,C 180,E1 -19430.404,E2 -19430.404} C_VEL
LIN {X 0,Y 242.398,Z 314.916,A -85,B 0,C 180,E1 -19433.34,E2 -19433.34} C_VEL
LIN {X 0,Y 242.634,Z 314.888,A -85,B 0,C 180,E1 -19438.34,E2 -19438.34} C_VEL
LIN {X 0,Y 242.633,Z 314.887,A -85,B 0,C 180,E1 -19441.66,E2 -19441.66} C_VEL
LIN {X 0,Y 242.403,Z 314.915,A -85,B 0,C 180,E1 -19446.66,E2 -19446.66} C_VEL
LIN {X 0,Y 242.267,Z 314.934,A -85,B 0,C 180,E1 -19450.024,E2 -19450.024} C_VEL
LIN {X 0,Y 242.166,Z 314.948,A -85,B 0,C 180,E1 -19455.141,E2 -19455.141} C_VEL
LIN {X 0,Y 242.071,Z 314.958,A -85,B 0,C 180,E1 -19458.624,E2 -19458.624} C_VEL
LIN {X 0,Y 242.006,Z 314.965,A -85,B 0,C 180,E1 -19462.18,E2 -19462.18} C_VEL
LIN {X 0,Y 242.066,Z 314.959,A -85,B 0,C 180,E1 -19465.838,E2 -19465.838} C_VEL
LIN {X 0,Y 242.007,Z 314.97,A -85,B 0,C 180,E1 -19469.583,E2 -19469.583} C_VEL
LIN {X 0,Y 242.26,Z 316.837,A -85,B 0,C 180,E1 -19473.449,E2 -19473.449} C_VEL
LIN {X 0,Y 242.498,Z 318.342,A -85,B 0,C 180,E1 -19476.048,E2 -19476.048} C_VEL
LIN {X 0,Y 241.875,Z 319.03,A -85,B 0,C 180,E1 -19476.96,E2 -19476.96} C_VEL
LIN {X 0,Y 239.17,Z 320.435,A -85,B 0,C 180,E1 -19478.388,E2 -19478.388} C_VEL
LIN {X 0,Y 236.493,Z 321.862,A -85,B 0,C 180,E1 -19479.848,E2 -19479.848} C_VEL
LIN {X 0,Y 235.948,Z 322.582,A -85,B 0,C 180,E1 -19480.793,E2 -19480.793} C_VEL
LIN {X 0,Y 236.114,Z 323.883,A -85,B 0,C 180,E1 -19482.738,E2 -19482.738} C_VEL
LIN {X 0,Y 237.212,Z 326.87,A -85,B 0,C 180,E1 -19483.167,E2 -19483.167} C_VEL
LIN {X 0,Y 239.299,Z 329.644,A -85,B 0,C 180,E1 -19483.836,E2 -19483.836} C_VEL
LIN {X 0,Y 241.242,Z 333.352,A -85,B 0,C 180,E1 -19484.507,E2 -19484.507} C_VEL
LIN {X 0,Y 245.846,Z 342.744,A -85,B 0,C 180,E1 -19486.205,E2 -19486.205} C_VEL
LIN {X 0,Y 250.025,Z 353.592,A -85,B 0,C 180,E1 -19487.999,E2 -19487.999} C_VEL
LIN {X 0,Y 253.662,Z 365.945,A -85,B 0,C 180,E1 -19489.973,E2 -19489.973} C_VEL
LIN {X 0,Y 256.066,Z 377.374,A -85,B 0,C 180,E1 -19491.792,E2 -19491.792} C_VEL
LIN {X 0,Y 257.47,Z 387.397,A -85,B 0,C 180,E1 -19493.448,E2 -19493.448} C_VEL
LIN {X 0,Y 258.226,Z 397.238,A -85,B 0,C 180,E1 -19495.142,E2 -19495.142} C_VEL
LIN {X 0,Y 256.255,Z 405.176,A -85,B 0,C 180,E1 -19496.268,E2 -19496.268} C_VEL
LIN {X 0,Y 252.424,Z 417.546,A -85,B 0,C 180,E1 -19498.297,E2 -19498.297} C_VEL
LIN {X 0,Y 248.375,Z 429.696,A -85,B 0,C 180,E1 -19500.784,E2 -19500.784} C_VEL
LIN {X 0,Y 245.102,Z 439.07,A -85,B 0,C 180,E1 -19503.153,E2 -19503.153} C_VEL
LIN {X 0,Y 242.174,Z 447.055,A -85,B 0,C 180,E1 -19505.572,E2 -19505.572} C_VEL
LIN {X 0,Y 239.316,Z 454.947,A -85,B 0,C 180,E1 -19508.464,E2 -19508.464} C_VEL
LIN {X 0,Y 236.614,Z 462.431,A -85,B 0,C 180,E1 -19511.892,E2 -19511.892} C_VEL
LIN {X 0,Y 234.866,Z 468.16,A -85,B 0,C 180,E1 -19515.265,E2 -19515.265} C_VEL
LIN {X 0,Y 233.809,Z 471.635,A -85,B 0,C 180,E1 -19517.853,E2 -19517.853} C_VEL
LIN {X 0,Y 233.036,Z 475.146,A -85,B 0,C 180,E1 -19521.327,E2 -19521.327} C_VEL
LIN {X 0,Y 232.686,Z 477.454,A -85,B 0,C 180,E1 -19524.801,E2 -19524.801} C_VEL
LIN {X 0,Y 232.644,Z 478.614,A -85,B 0,C 180,E1 -19528.268,E2 -19528.268} C_VEL
LIN {X 0,Y 232.715,Z 478.767,A -85,B 0,C 180,E1 -19529.999,E2 -19529.999} C_VEL
LIN {X 0,Y 232.626,Z 478.163,A -85,B 0,C 180,E1 -19533.463,E2 -19533.463} C_VEL
LIN {X 0,Y 232.807,Z 476.418,A -85,B 0,C 180,E1 -19536.935,E2 -19536.935} C_VEL
LIN {X 0,Y 233.378,Z 473.505,A -85,B 0,C 180,E1 -19540.409,E2 -19540.409} C_VEL
LIN {X 0,Y 234.479,Z 469.358,A -85,B 0,C 180,E1 -19543.873,E2 -19543.873} C_VEL
LIN {X 0,Y 236.213,Z 463.864,A -85,B 0,C 180,E1 -19547.308,E2 -19547.308} C_VEL
